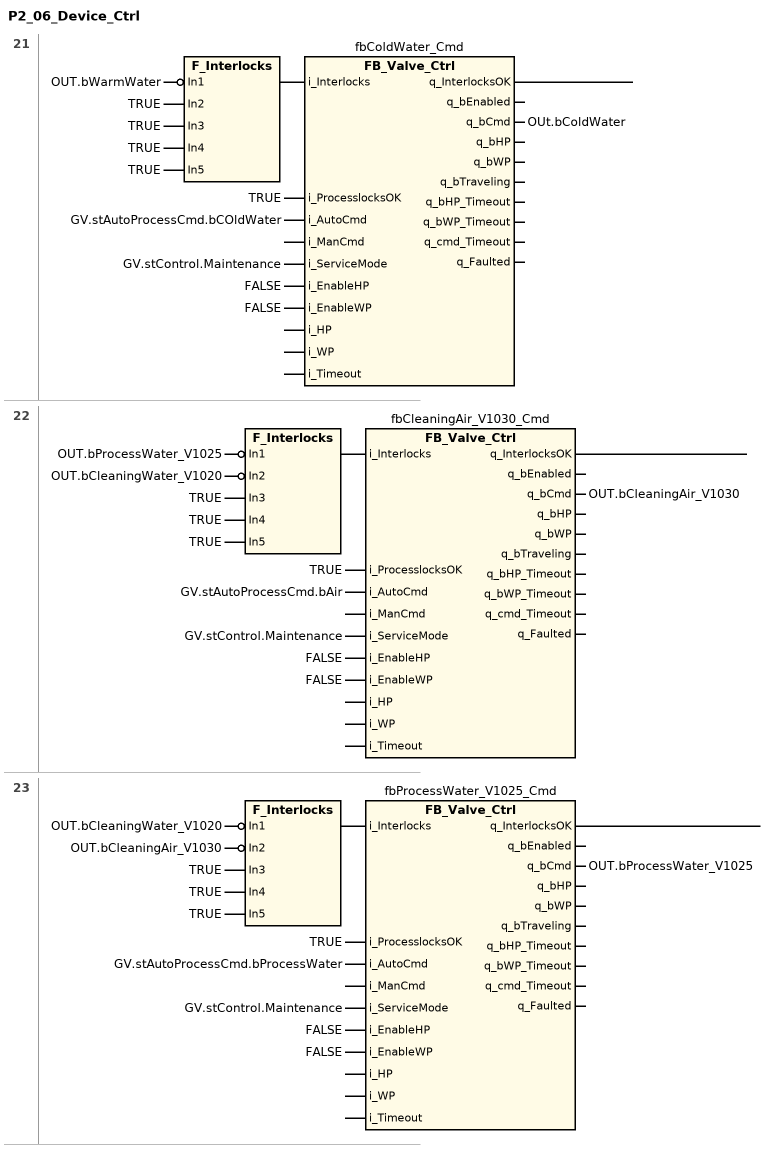
// NETWORK 21
fbColdWater_Cmd(
    i_Interlocks := F_Interlocks(In1 := NOT OUT.bWarmWater, In2 := TRUE, In3 := TRUE, In4 := TRUE, In5 := TRUE),
    i_ProcesslocksOK := TRUE,
    i_AutoCmd := GV.stAutoProcessCmd.bCOldWater,
    i_ServiceMode := GV.stControl.Maintenance,
    i_EnableHP := FALSE,
    i_EnableWP := FALSE,
    q_bCmd => OUt.bColdWater); // FB_Valve_Ctrl

// NETWORK 22
fbCleaningAir_V1030_Cmd(
    i_Interlocks := F_Interlocks(In1 := NOT OUT.bProcessWater_V1025, In2 := NOT OUT.bCleaningWater_V1020, In3 := TRUE, In4 := TRUE, In5 := TRUE),
    i_ProcesslocksOK := TRUE,
    i_AutoCmd := GV.stAutoProcessCmd.bAir,
    i_ServiceMode := GV.stControl.Maintenance,
    i_EnableHP := FALSE,
    i_EnableWP := FALSE,
    q_bCmd => OUT.bCleaningAir_V1030); // FB_Valve_Ctrl

// NETWORK 23
fbProcessWater_V1025_Cmd(
    i_Interlocks := F_Interlocks(In1 := NOT OUT.bCleaningWater_V1020, In2 := NOT OUT.bCleaningAir_V1030, In3 := TRUE, In4 := TRUE, In5 := TRUE),
    i_ProcesslocksOK := TRUE,
    i_AutoCmd := GV.stAutoProcessCmd.bProcessWater,
    i_ServiceMode := GV.stControl.Maintenance,
    i_EnableHP := FALSE,
    i_EnableWP := FALSE,
    q_bCmd => OUT.bProcessWater_V1025); // FB_Valve_Ctrl

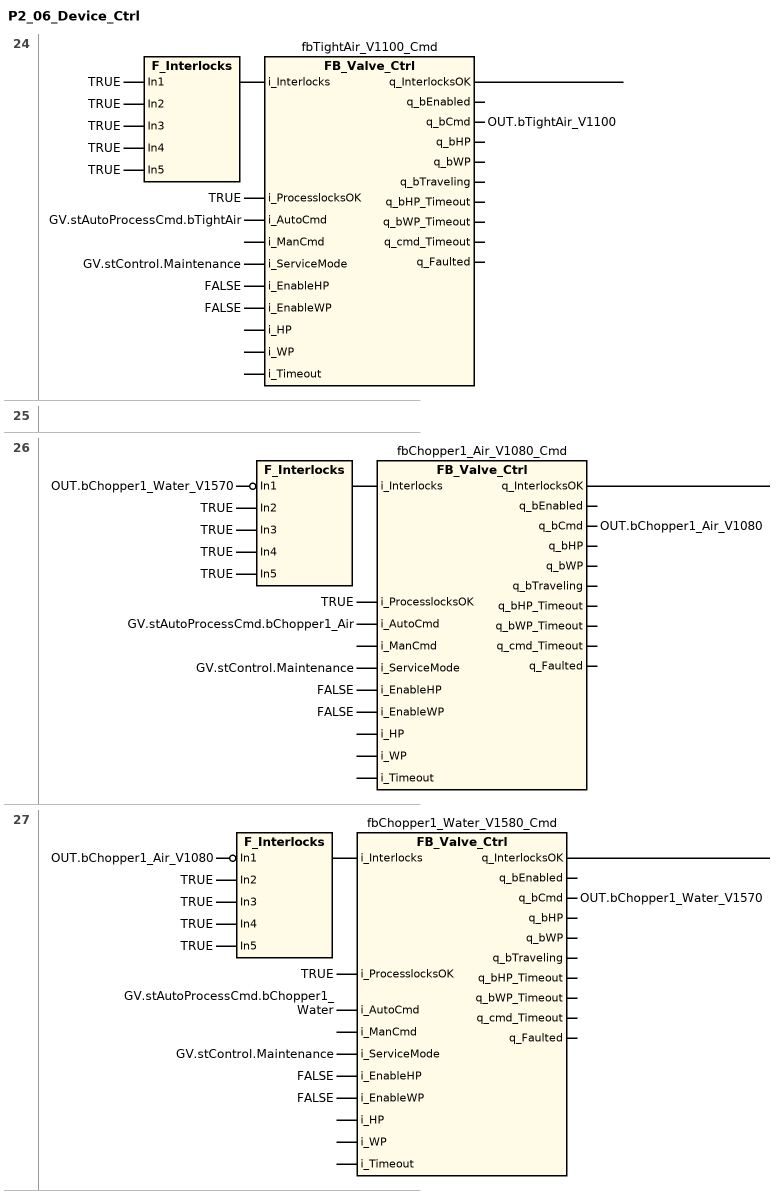
// NETWORK 24
fbTightAir_V1100_Cmd(
    i_Interlocks := F_Interlocks(In1 := TRUE, In2 := TRUE, In3 := TRUE, In4 := TRUE, In5 := TRUE),
    i_ProcesslocksOK := TRUE,
    i_AutoCmd := GV.stAutoProcessCmd.bTightAir,
    i_ServiceMode := GV.stControl.Maintenance,
    i_EnableHP := FALSE,
    i_EnableWP := FALSE,
    q_bCmd => OUT.bTightAir_V1100); // FB_Valve_Ctrl

// NETWORK 25

// NETWORK 26
fbChopper1_Air_V1080_Cmd(
    i_Interlocks := F_Interlocks(In1 := NOT OUT.bChopper1_Water_V1570, In2 := TRUE, In3 := TRUE, In4 := TRUE, In5 := TRUE),
    i_ProcesslocksOK := TRUE,
    i_AutoCmd := GV.stAutoProcessCmd.bChopper1_Air,
    i_ServiceMode := GV.stControl.Maintenance,
    i_EnableHP := FALSE,
    i_EnableWP := FALSE,
    q_bCmd => OUT.bChopper1_Air_V1080); // FB_Valve_Ctrl

// NETWORK 27
fbChopper1_Water_V1580_Cmd(
    i_Interlocks := F_Interlocks(In1 := NOT OUT.bChopper1_Air_V1080, In2 := TRUE, In3 := TRUE, In4 := TRUE, In5 := TRUE),
    i_ProcesslocksOK := TRUE,
    i_AutoCmd := GV.stAutoProcessCmd.bChopper1_Water,
    i_ServiceMode := GV.stControl.Maintenance,
    i_EnableHP := FALSE,
    i_EnableWP := FALSE,
    q_bCmd => OUT.bChopper1_Water_V1570); // FB_Valve_Ctrl

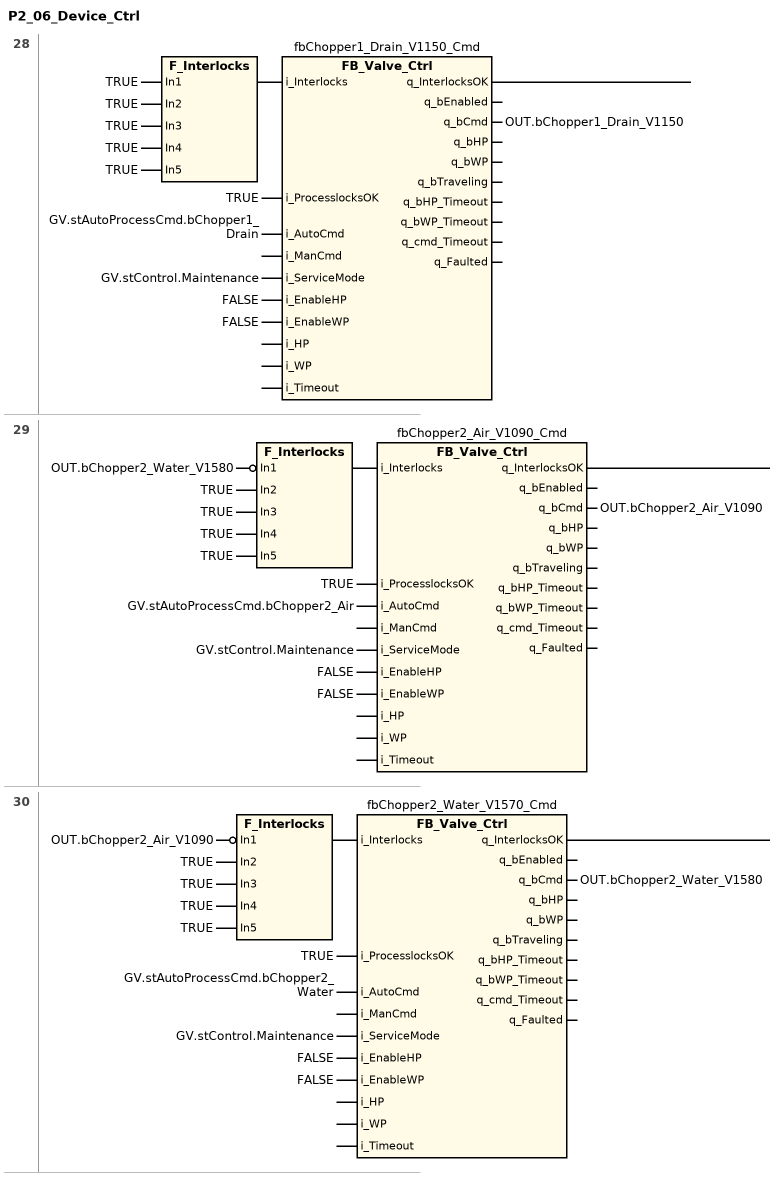
// NETWORK 28
fbChopper1_Drain_V1150_Cmd(
    i_Interlocks := F_Interlocks(In1 := TRUE, In2 := TRUE, In3 := TRUE, In4 := TRUE, In5 := TRUE),
    i_ProcesslocksOK := TRUE,
    i_AutoCmd := GV.stAutoProcessCmd.bChopper1_Drain,
    i_ServiceMode := GV.stControl.Maintenance,
    i_EnableHP := FALSE,
    i_EnableWP := FALSE,
    q_bCmd => OUT.bChopper1_Drain_V1150); // FB_Valve_Ctrl

// NETWORK 29
fbChopper2_Air_V1090_Cmd(
    i_Interlocks := F_Interlocks(In1 := NOT OUT.bChopper2_Water_V1580, In2 := TRUE, In3 := TRUE, In4 := TRUE, In5 := TRUE),
    i_ProcesslocksOK := TRUE,
    i_AutoCmd := GV.stAutoProcessCmd.bChopper2_Air,
    i_ServiceMode := GV.stControl.Maintenance,
    i_EnableHP := FALSE,
    i_EnableWP := FALSE,
    q_bCmd => OUT.bChopper2_Air_V1090); // FB_Valve_Ctrl

// NETWORK 30
fbChopper2_Water_V1570_Cmd(
    i_Interlocks := F_Interlocks(In1 := NOT OUT.bChopper2_Air_V1090, In2 := TRUE, In3 := TRUE, In4 := TRUE, In5 := TRUE),
    i_ProcesslocksOK := TRUE,
    i_AutoCmd := GV.stAutoProcessCmd.bChopper2_Water,
    i_ServiceMode := GV.stControl.Maintenance,
    i_EnableHP := FALSE,
    i_EnableWP := FALSE,
    q_bCmd => OUT.bChopper2_Water_V1580); // FB_Valve_Ctrl

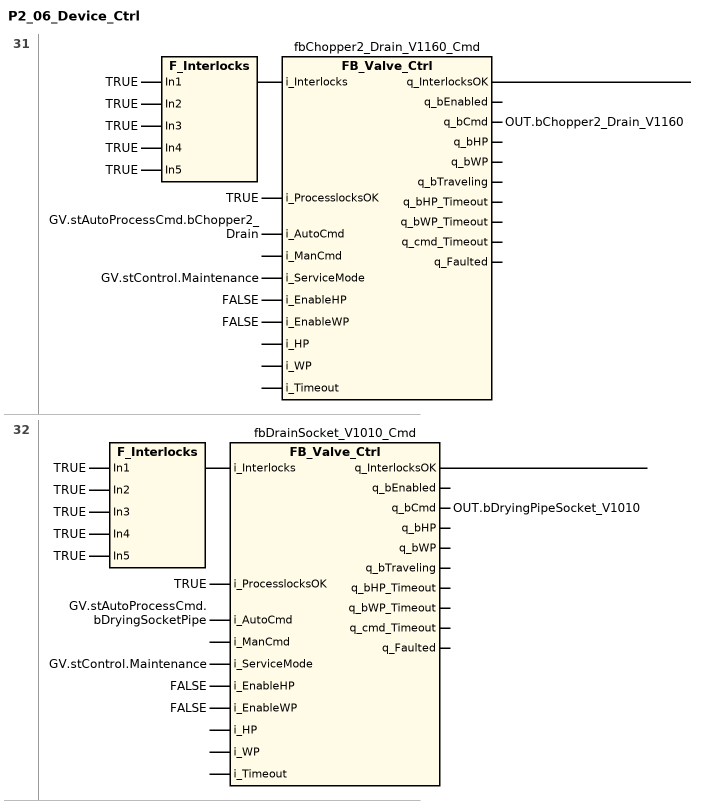
// NETWORK 31
fbChopper2_Drain_V1160_Cmd(
    i_Interlocks := F_Interlocks(In1 := TRUE, In2 := TRUE, In3 := TRUE, In4 := TRUE, In5 := TRUE),
    i_ProcesslocksOK := TRUE,
    i_AutoCmd := GV.stAutoProcessCmd.bChopper2_Drain,
    i_ServiceMode := GV.stControl.Maintenance,
    i_EnableHP := FALSE,
    i_EnableWP := FALSE,
    q_bCmd => OUT.bChopper2_Drain_V1160); // FB_Valve_Ctrl

// NETWORK 32
fbDrainSocket_V1010_Cmd(
    i_Interlocks := F_Interlocks(In1 := TRUE, In2 := TRUE, In3 := TRUE, In4 := TRUE, In5 := TRUE),
    i_ProcesslocksOK := TRUE,
    i_AutoCmd := GV.stAutoProcessCmd.bDryingSocketPipe,
    i_ServiceMode := GV.stControl.Maintenance,
    i_EnableHP := FALSE,
    i_EnableWP := FALSE,
    q_bCmd => OUT.bDryingPipeSocket_V1010); // FB_Valve_Ctrl

END_PROGRAM

// ---- FB/FB_Valve53_Ctrl.TcPOU
FUNCTION_BLOCK FB_Valve53_Ctrl
VAR_INPUT
	i_bInterlock		:BOOL;
	i_bProcesslock		:BOOL;
	i_bCmd_Disable		:BOOL;
	i_bCmd_Close		:BOOL;
	i_bCmd_HalfOpen		:BOOL;
	i_bCmd_Open			:BOOL;
	i_bSensorClosed		:BOOL;
	i_bSensorHalfOpen	:BOOL;
	i_bSensorOpen		:BOOL;
	i_tTimeout			:TIME;
	i_tTimeOutHalf		:TIME;
END_VAR
VAR_OUTPUT
	q_bCmd_Release		:BOOL;
	q_bCmd_Close		:BOOL;
	q_bCmd_Open			:BOOL;
	q_bEnabled			:BOOL;
	q_bClosed			:BOOL;
	q_bHalfOpened		:BOOL;
	q_bOpened			:BOOL;
	q_bTraveling		:BOOL;
	q_bClose_Timeout	:BOOL;
	q_bOpen_Timeout		:BOOL;
	q_bHOpen_Timeout	:BOOL;
END_VAR
VAR
	tonTimeoutClose		:TON;
	tonTimeOutHOpen		:TON;
	tonTimeoutOpen		:TON;
	bMidPosReq			:BOOL;
END_VAR
VAR // added by the converter: edge detectors and wires of the graphical bodies
    _rt1, _rt2, _rt3 : R_TRIG;
    _w1, _w2, _w3, _w4, _w5 : BOOL;
END_VAR

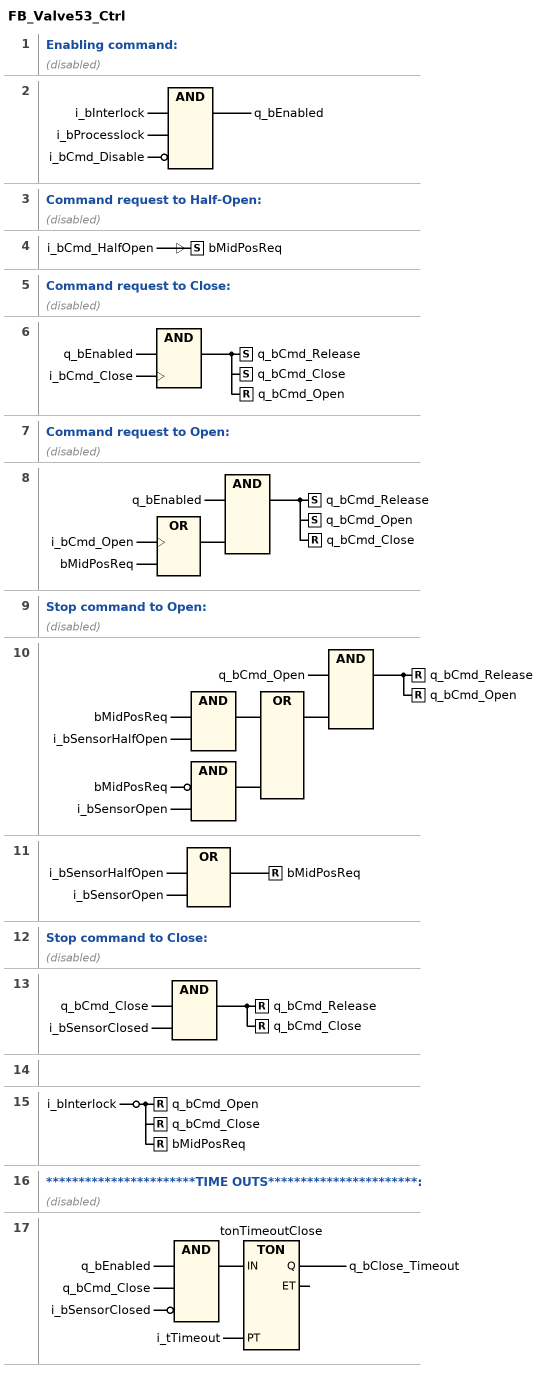
// NETWORK 1 (disabled)
// label: Enabling command

// NETWORK 2
q_bEnabled := i_bInterlock AND i_bProcesslock AND NOT i_bCmd_Disable;

// NETWORK 3 (disabled)
// label: Command request to Half-Open

// NETWORK 4
_rt1(CLK := i_bCmd_HalfOpen);
bMidPosReq S= _rt1.Q;

// NETWORK 5 (disabled)
// label: Command request to Close

// NETWORK 6
_rt2(CLK := i_bCmd_Close);
_w1 := q_bEnabled AND _rt2.Q;
q_bCmd_Release S= _w1;
q_bCmd_Close S= _w1;
q_bCmd_Open R= _w1;

// NETWORK 7 (disabled)
// label: Command request to Open

// NETWORK 8
_rt3(CLK := i_bCmd_Open);
_w2 := q_bEnabled AND (_rt3.Q OR bMidPosReq);
q_bCmd_Release S= _w2;
q_bCmd_Open S= _w2;
q_bCmd_Close R= _w2;

// NETWORK 9 (disabled)
// label: Stop command to Open

// NETWORK 10
_w3 := q_bCmd_Open AND (bMidPosReq AND i_bSensorHalfOpen OR NOT bMidPosReq AND i_bSensorOpen);
q_bCmd_Release R= _w3;
q_bCmd_Open R= _w3;

// NETWORK 11
bMidPosReq R= i_bSensorHalfOpen OR i_bSensorOpen;

// NETWORK 12 (disabled)
// label: Stop command to Close

// NETWORK 13
_w4 := q_bCmd_Close AND i_bSensorClosed;
q_bCmd_Release R= _w4;
q_bCmd_Close R= _w4;

// NETWORK 14

// NETWORK 15
_w5 := NOT i_bInterlock;
q_bCmd_Open R= _w5;
q_bCmd_Close R= _w5;
bMidPosReq R= _w5;

// NETWORK 16 (disabled)
// label: ***********************TIME OUTS***********************

// NETWORK 17
tonTimeoutClose(IN := q_bEnabled AND q_bCmd_Close AND NOT i_bSensorClosed, PT := i_tTimeout); // TON
q_bClose_Timeout := tonTimeoutClose.Q;

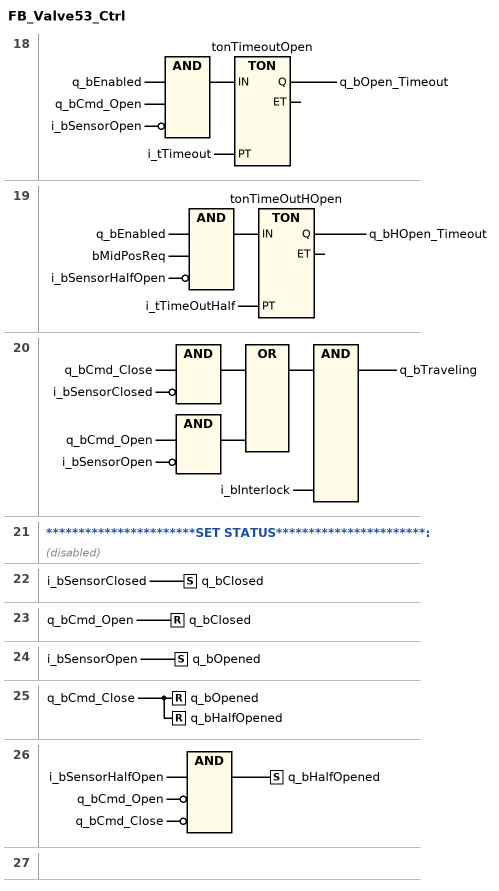
// NETWORK 18
tonTimeoutOpen(IN := q_bEnabled AND q_bCmd_Open AND NOT i_bSensorOpen, PT := i_tTimeout); // TON
q_bOpen_Timeout := tonTimeoutOpen.Q;

// NETWORK 19
tonTimeOutHOpen(IN := q_bEnabled AND bMidPosReq AND NOT i_bSensorHalfOpen, PT := i_tTimeOutHalf); // TON
q_bHOpen_Timeout := tonTimeOutHOpen.Q;

// NETWORK 20
q_bTraveling := (q_bCmd_Close AND NOT i_bSensorClosed OR q_bCmd_Open AND NOT i_bSensorOpen) AND i_bInterlock;

// NETWORK 21 (disabled)
// label: ***********************SET STATUS***********************

// NETWORK 22
q_bClosed S= i_bSensorClosed;

// NETWORK 23
q_bClosed R= q_bCmd_Open;

// NETWORK 24
q_bOpened S= i_bSensorOpen;

// NETWORK 25
q_bOpened R= q_bCmd_Close;
q_bHalfOpened R= q_bCmd_Close;

// NETWORK 26
q_bHalfOpened S= i_bSensorHalfOpen AND NOT q_bCmd_Open AND NOT q_bCmd_Close;

// NETWORK 27

END_FUNCTION_BLOCK

// ---- FB/FB_Mixer_Ctrl.TcPOU
FUNCTION_BLOCK FB_Mixer_Ctrl
VAR_INPUT
	i_Interlocks		:ARRAY[1..5] OF BOOL;
	i_AutoCmdFwd		:BOOL;
	i_AutoCmdBcw		:BOOL;
	i_AutoSpeedSP		:REAL;
	i_ManCmdFwd			:BOOL;
	i_ManCmdBcw			:BOOL;
	i_ManStop			:BOOL;
	i_ManSpeedSP		:REAL;
	i_SpeedAP			:REAL;
	i_CurrentAP			:REAL;
	i_ServiceMode		:BOOL;
END_VAR
VAR_OUTPUT
	q_InterlocksOK		:BOOL;
	q_bCmdFwd			:BOOL;
	q_bCmdBcw			:BOOL;
	q_rSpeedSP			:REAL;
END_VAR
VAR
	bCmdFwd				:BOOL;
	bCmdBcw				:BOOL;
	tofCMDFwd			:TOF;
	tofCMDBcw			:TOF;
	tonFwdOff			:TON;
	tonBcwOff			:TON;
END_VAR
VAR // added by the converter: edge detectors and wires of the graphical bodies
    _w1 : BOOL;
END_VAR

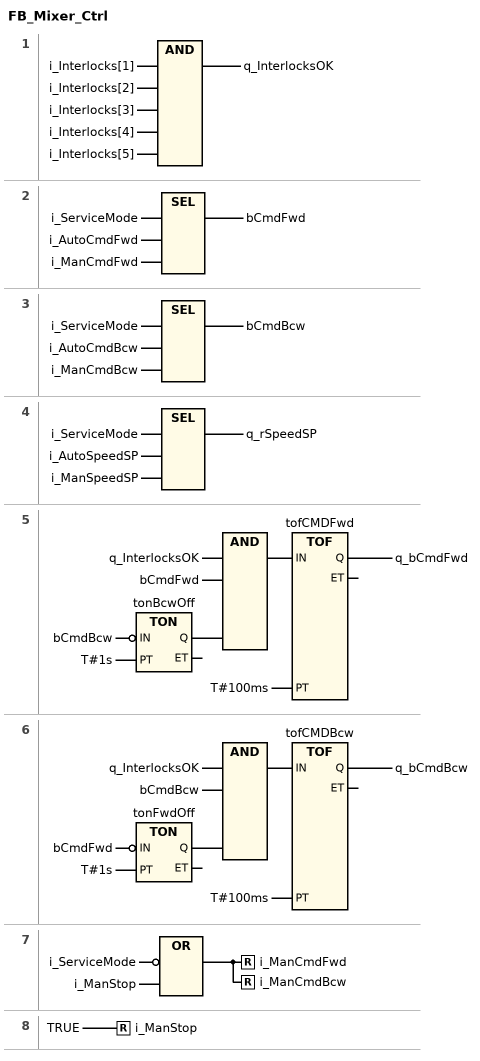
// NETWORK 1
q_InterlocksOK := i_Interlocks[1] AND i_Interlocks[2] AND i_Interlocks[3] AND i_Interlocks[4] AND i_Interlocks[5];

// NETWORK 2
bCmdFwd := SEL(i_ServiceMode, i_AutoCmdFwd, i_ManCmdFwd);

// NETWORK 3
bCmdBcw := SEL(i_ServiceMode, i_AutoCmdBcw, i_ManCmdBcw);

// NETWORK 4
q_rSpeedSP := SEL(i_ServiceMode, i_AutoSpeedSP, i_ManSpeedSP);

// NETWORK 5
tonBcwOff(IN := NOT bCmdBcw, PT := T#1s); // TON
tofCMDFwd(IN := q_InterlocksOK AND bCmdFwd AND tonBcwOff.Q, PT := T#100ms); // TOF
q_bCmdFwd := tofCMDFwd.Q;

// NETWORK 6
tonFwdOff(IN := NOT bCmdFwd, PT := T#1s); // TON
tofCMDBcw(IN := q_InterlocksOK AND bCmdBcw AND tonFwdOff.Q, PT := T#100ms); // TOF
q_bCmdBcw := tofCMDBcw.Q;

// NETWORK 7
_w1 := NOT i_ServiceMode OR i_ManStop;
i_ManCmdFwd R= _w1;
i_ManCmdBcw R= _w1;

// NETWORK 8
i_ManStop R= TRUE;

END_FUNCTION_BLOCK

// ---- FB/FB_AnalogOutput.TcPOU
// Created by Dimitar Stojanov 06.2023 

//Functionality: Use this block to scale Analog Outputs

FUNCTION_BLOCK FB_AnalogOutput
VAR_INPUT
	i_rValue 							:REAL;
	i_rData_Low 						:REAL;
	i_rData_High 						:REAL;
	i_rScaled_Low						:INT	:=0;
	i_rScaled_High						:INT	:=32676;
	i_iOffset 							:INT;
	
END_VAR
VAR_OUTPUT
	q_iScaled							:INT;
END_VAR
VAR
	K								    :REAL;
END_VAR

K := ((i_rScaled_High - i_rScaled_Low) / (i_rData_High - i_rData_Low));
q_iScaled:=REAL_TO_INT((K * i_rValue) + i_iOffset);

END_FUNCTION_BLOCK

// ---- FB/FB_Chopper_Ctrl.TcPOU
FUNCTION_BLOCK FB_Chopper_Ctrl
VAR_INPUT
	i_Interlocks		:ARRAY[1..5] OF BOOL;
	i_AutoSlowCmd		:BOOL;
	i_AutoFastCmd		:BOOL;
	i_ManSlowCmd		:BOOL;
	i_ManFastCmd		:BOOL;
	I_ManStop			:BOOL;
	i_rSpeed			:REAL;
	i_ServiceMode		:BOOL;
END_VAR
VAR_OUTPUT
	q_InterlocksOK		:BOOL;
	q_bCmdFast			:BOOL;
	q_bCmdSlow			:BOOL;
	q_rSpeed			:REAL;
END_VAR
VAR
	bCmdSlow			:BOOL;
	bCmdFast			:BOOL;
	tofSlowCMD			:TOF;
	tofFastCMD			:TOF;
	tonSlowOff			:TON;
	tonFastOff			:TON;
END_VAR
VAR // added by the converter: edge detectors and wires of the graphical bodies
    _w1 : BOOL;
END_VAR

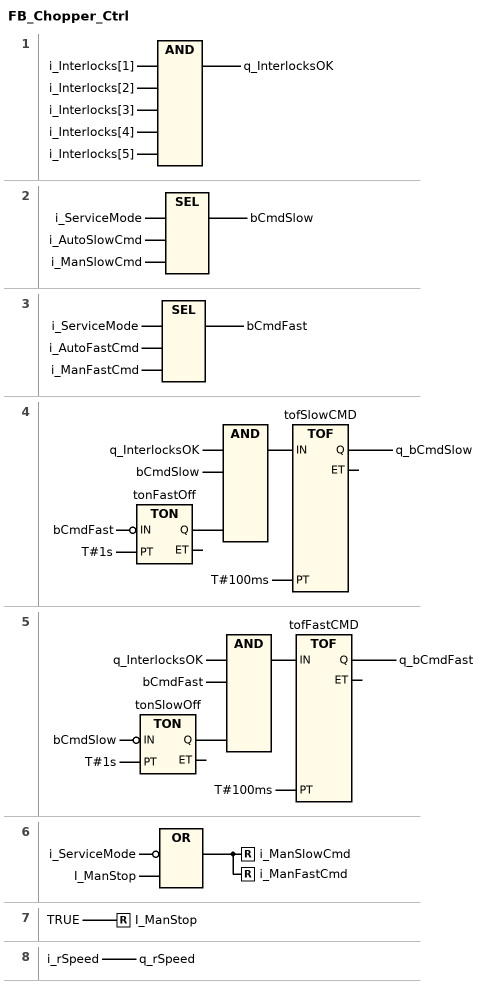
// NETWORK 1
q_InterlocksOK := i_Interlocks[1] AND i_Interlocks[2] AND i_Interlocks[3] AND i_Interlocks[4] AND i_Interlocks[5];

// NETWORK 2
bCmdSlow := SEL(i_ServiceMode, i_AutoSlowCmd, i_ManSlowCmd);

// NETWORK 3
bCmdFast := SEL(i_ServiceMode, i_AutoFastCmd, i_ManFastCmd);

// NETWORK 4
tonFastOff(IN := NOT bCmdFast, PT := T#1s); // TON
tofSlowCMD(IN := q_InterlocksOK AND bCmdSlow AND tonFastOff.Q, PT := T#100ms); // TOF
q_bCmdSlow := tofSlowCMD.Q;

// NETWORK 5
tonSlowOff(IN := NOT bCmdSlow, PT := T#1s); // TON
tofFastCMD(IN := q_InterlocksOK AND bCmdFast AND tonSlowOff.Q, PT := T#100ms); // TOF
q_bCmdFast := tofFastCMD.Q;

// NETWORK 6
_w1 := NOT i_ServiceMode OR I_ManStop;
i_ManSlowCmd R= _w1;
i_ManFastCmd R= _w1;

// NETWORK 7
I_ManStop R= TRUE;

// NETWORK 8
q_rSpeed := i_rSpeed;

END_FUNCTION_BLOCK

// ---- FB/FB_Valve_Ctrl.TcPOU
FUNCTION_BLOCK FB_Valve_Ctrl
VAR_INPUT
	i_Interlocks		:ARRAY[1..5] OF BOOL;
	i_ProcesslocksOK	:BOOL;
	i_AutoCmd			:BOOL;
	i_ManCmd			:BOOL;
	i_ServiceMode		:BOOL;
	i_EnableHP			:BOOL;
	i_EnableWP			:BOOL;
	i_HP				:BOOL;
	i_WP				:BOOL;
	i_Timeout			:TIME;
END_VAR
VAR_OUTPUT
	q_InterlocksOK		:BOOL;
	q_bEnabled			:BOOL;
	q_bCmd				:BOOL;
	q_bHP				:BOOL;
	q_bWP				:BOOL;
	q_bTraveling		:BOOL;
	q_bHP_Timeout		:BOOL;
	q_bWP_Timeout		:BOOL;
	q_cmd_Timeout		:BOOL;
	q_Faulted			:BOOL;
END_VAR
VAR
	tonTimeoutHP		:TON;
	tonTimeoutWP		:TON;
	tonTimeoutCmd		:TON;
	tofDelayOut			:TOF;
	bCmd				:BOOL;
END_VAR

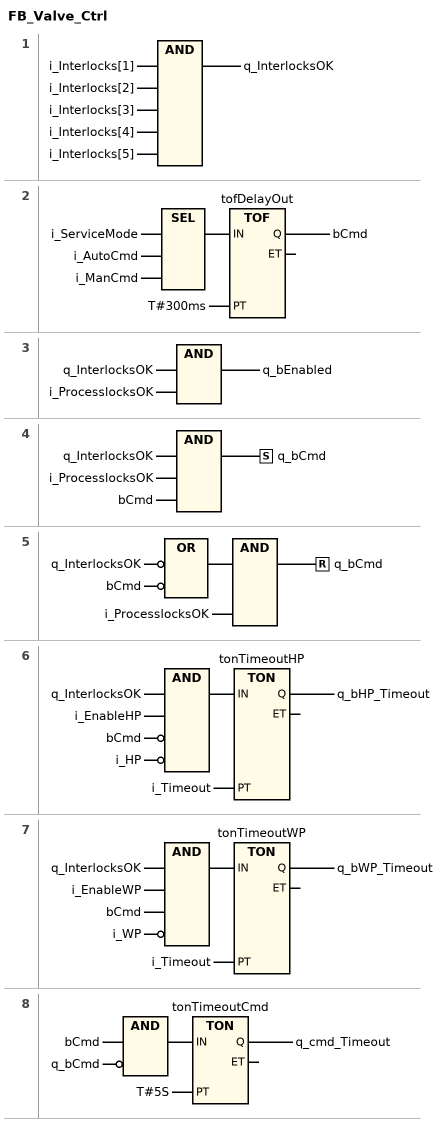
// NETWORK 1
q_InterlocksOK := i_Interlocks[1] AND i_Interlocks[2] AND i_Interlocks[3] AND i_Interlocks[4] AND i_Interlocks[5];

// NETWORK 2
tofDelayOut(IN := SEL(i_ServiceMode, i_AutoCmd, i_ManCmd), PT := T#300ms); // TOF
bCmd := tofDelayOut.Q;

// NETWORK 3
q_bEnabled := q_InterlocksOK AND i_ProcesslocksOK;

// NETWORK 4
q_bCmd S= q_InterlocksOK AND i_ProcesslocksOK AND bCmd;

// NETWORK 5
q_bCmd R= (NOT q_InterlocksOK OR NOT bCmd) AND i_ProcesslocksOK;

// NETWORK 6
tonTimeoutHP(IN := q_InterlocksOK AND i_EnableHP AND NOT bCmd AND NOT i_HP, PT := i_Timeout); // TON
q_bHP_Timeout := tonTimeoutHP.Q;

// NETWORK 7
tonTimeoutWP(IN := q_InterlocksOK AND i_EnableWP AND bCmd AND NOT i_WP, PT := i_Timeout); // TON
q_bWP_Timeout := tonTimeoutWP.Q;

// NETWORK 8
tonTimeoutCmd(IN := bCmd AND NOT q_bCmd, PT := T#5S); // TON
q_cmd_Timeout := tonTimeoutCmd.Q;

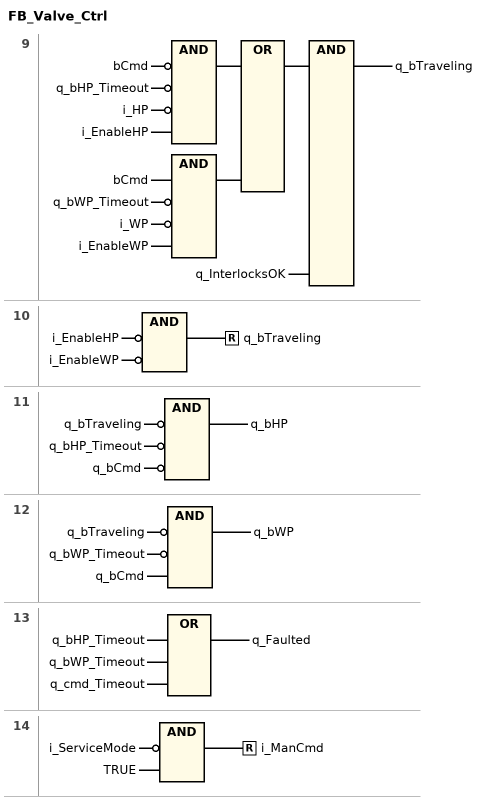
// NETWORK 9
q_bTraveling := (NOT bCmd AND NOT q_bHP_Timeout AND NOT i_HP AND i_EnableHP OR bCmd AND NOT q_bWP_Timeout AND NOT i_WP AND i_EnableWP) AND q_InterlocksOK;

// NETWORK 10
q_bTraveling R= NOT i_EnableHP AND NOT i_EnableWP;

// NETWORK 11
q_bHP := NOT q_bTraveling AND NOT q_bHP_Timeout AND NOT q_bCmd;

// NETWORK 12
q_bWP := NOT q_bTraveling AND NOT q_bWP_Timeout AND q_bCmd;

// NETWORK 13
q_Faulted := q_bHP_Timeout OR q_bWP_Timeout OR q_cmd_Timeout;

// NETWORK 14
i_ManCmd R= NOT i_ServiceMode AND TRUE;

END_FUNCTION_BLOCK

// ---- POUs/2. Process/Production/_Discharging.TcPOU
PROGRAM _Discharging
VAR_INPUT
	i_bStart							:BOOL;
	i_bProcessFinished					:BOOL;
	i_bStepFinished						:BOOL;
	i_bSkipStep							:BOOL;
	i_bBarrelInPos						:BOOL;
	i_bManualFlapOpen					:BOOL;
	i_bManualFlapClose					:BOOL;
	i_iMixer							:INT;
	i_rMixerSpeed						:REAL;
	i_bMixerStart						:BOOL; 	
	i_iChopper							:INT;	
END_VAR
VAR
	iStep						:INT;
	iPrevStep					:INT;
	Seq_TON						:ARRAY[0..9] OF TON;
	Seq_Time					:ARRAY[0..9] OF TIME;
	trigMixer					:R_TRIG;
	bStartMixer					:BOOL;
	tonStepTime					:TON;
END_VAR
VAR_OUTPUT
	q_bRunning						:BOOL;
	q_bFinished						:BOOL;
	q_stCmd							:ST_ProcessCmd;
	q_bDisOpenReq					:BOOL;
	q_bDischargeCmdEnable			:BOOL;
	q_bBarrelInPosReq				:BOOL;
	q_tStepTime						:TIME;
END_VAR

trigMixer(CLK:=i_bMixerStart);


q_bRunning:=iStep<>0;

IF i_bSkipStep THEN
	iStep:=1000;
END_IF

IF NOT i_bStart THEN
	iStep:=0;
END_IF

CASE iStep OF
	0:
		IF i_bStart THEN
			q_bFinished:=FALSE;
			iStep:=40;
		END_IF
		
		IF iStep <> 0 THEN
			iPrevStep:=0;
		END_IF
		
	40:
		IF i_bBarrelInPos THEN
			iStep:=50;
		END_IF
		
	50:
		IF i_bManualFlapOpen THEN
			iStep:=100;
		END_IF
		
		IF iStep <> 50 THEN
			iPrevStep:=50;
		END_IF
	
	100:
		
		IF i_bProcessFinished THEN
			iStep:=1000;
		END_IF
		IF iStep <> 100 THEN
			iPrevStep:=100;
		END_IF

		
	1000:
		q_bFinished:=TRUE;
		IF i_bStepFinished THEN
			iStep:=0;
		END_IF
END_CASE

IF trigMixer.Q THEN
	bStartMixer:= NOT bStartMixer;
END_IF

q_bBarrelInPosReq:=F_StepCMP(iStep,40,0,0,0,0,0,0,0,0,0);

q_bDisOpenReq:=F_StepCMP(iStep,50,0,0,0,0,0,0,0,0,0);
IF F_StepCMP(iStep,50,0,0,0,0,0,0,0,0,0) THEN
	q_stCmd.bDischargeClose:=FALSE;
	q_stCmd.bDischargeOpen:=TRUE;
ELSE
	q_stCmd.bDischargeClose:=FALSE;
	q_stCmd.bDischargeOpen:=FALSE;
END_IF

q_bDischargeCmdEnable:=F_StepCMP(iStep,100,0,0,0,0,0,0,0,0,0);

IF F_StepCMP(iStep,100,0,0,0,0,0,0,0,0,0) AND bStartMixer THEN
	q_stCmd.iMixer:=i_iMixer;
	q_stCmd.rMixerSpeed:=i_rMixerSpeed;
ELSE
	q_stCmd.iMixer:=0;
	q_stCmd.rMixerSpeed:=0;
	bStartMixer:=FALSE;
END_IF

IF F_StepCMP(iStep,100,0,0,0,0,0,0,0,0,0) AND bStartMixer THEN
	q_stCmd.iChopper:=i_iChopper;
ELSE
	q_stCmd.iChopper:=0;
END_IF

q_stCmd.bTightAir:=F_StepCMP(iStep,50,100,0,0,0,0,0,0,0,0);
q_stCmd.bChopper1_Air:=F_StepCMP(iStep,50,100,0,0,0,0,0,0,0,0);
q_stCmd.bChopper2_Air:=F_StepCMP(iStep,50,100,0,0,0,0,0,0,0,0);

//Statistic and Status
tonStepTime(IN:=q_bRunning,PT:=T#5H);
q_tStepTime:=tonStepTime.ET;

END_PROGRAM

// ---- FB/F_StepCMP.TcPOU
FUNCTION F_StepCMP : BOOL
VAR_INPUT
	iStep			:INT:=0;
	i1				:INT:=0;
	i2				:INT:=0;
	i3				:INT:=0;
	i4				:INT:=0;
	i5				:INT:=0;
	i6				:INT:=0;
	i7				:INT:=0;
	i8				:INT:=0;
	i9				:INT:=0;
	i10				:INT:=0;
END_VAR

F_StepCMP:=((iStep=i1) OR 
			(iStep=i2) OR 
			(iStep=i3) OR 
			(iStep=i4) OR 
			(iStep=i5) OR 
			(iStep=i6) OR 
			(iStep=i7) OR 
			(iStep=i8) OR 
			(iStep=i9) OR 
			(iStep=i10)) AND
			(iStep<>0);

END_FUNCTION

// ---- FB/F_Interlocks.TcPOU
FUNCTION F_Interlocks : ARRAY[1..5] OF BOOL
VAR_INPUT
	In1		:BOOL;
	In2		:BOOL;
	In3		:BOOL;
	In4		:BOOL;
	In5		:BOOL;
END_VAR
VAR
END_VAR

F_Interlocks[1] := In1;
F_Interlocks[2] := In2;
F_Interlocks[3] := In3;
F_Interlocks[4] := In4;
F_Interlocks[5] := In5;

END_FUNCTION

// ---- POUs/3. Report/P3_06_CreateReport.TcPOU
PROGRAM P3_06_CreateReport
VAR
	iStep					:INT;
	iError					:INT;
	tonResetError			:TON;
	trigStart				:R_TRIG;
	tonDelayStart			:TON;
	
	
	
	fbReport				:FB_PythonScript;
	fbSettingDelete			:FB_FileDelete;
	fbRecipeDelete			:FB_FileDelete;
	fbDeleteOldestBatch		:FB_DeleteOldestFile;
	fbSaveAsAlarm			:FB_FileSaveAs;
END_VAR


VAR PERSISTENT
	iReportsCreated			:INT;
END_VAR

ACT_CMDs();
tonResetError(IN:=(iError<>0),PT:=T#3S);
IF tonResetError.Q THEN
	iError:=0;
END_IF

trigStart(CLK:=GV.bBatchClose);

tonDelayStart(IN:=(iStep=10),PT:=T#1S);
CASE iStep OF
	
	0:
		IF trigStart.Q THEN
			iError:=0;
			iStep:=10;
		END_IF
		
	10:
		IF tonDelayStart.Q THEN
			iStep:=20;
		END_IF
		
	20:
		GV.stReport.bExport_Alarms:=TRUE;
		iStep:=25;
	25:
		IF NOT GV.stReport.bExport_Alarms THEN
			iStep:=30;
		END_IF
	26:
		GV.stReport.bSaveAs_Alarms:=TRUE;
		iStep:=27;
	27:
		IF NOT fbSaveAsAlarm.q_bBusy THEN
			iStep:=30;
		END_IF
		
	30:
		GV.stReport.bCreate_Report:=TRUE;
		IF fbReport.q_bBusy THEN
			iStep:=35;
		END_IF
	35:
		IF NOT fbReport.q_bBusy AND fbReport.q_bDone THEN
			iStep:=40;
		ELSIF fbReport.q_bError THEN
			iError:=iStep;
			iStep:=999;
		END_IF
	40:
		GV.stReport.bDelete_Data:=TRUE;
		iStep:=45;
	45:
		IF NOT GV.stReport.bDelete_Data THEN
			iStep:=50;
		END_IF
		
	50:
		GV.stReport.bDelete_OldestReport:=TRUE;
		IF fbDeleteOldestBatch.q_bBusy THEN
			iStep:=55;
		END_IF
	55:
		IF NOT fbDeleteOldestBatch.q_bBusy AND fbDeleteOldestBatch.q_bDone THEN
			iStep:=900;
		ELSIF fbDeleteOldestBatch.q_bError THEN
			iStep:=900;
			iError:=iStep;
		END_IF
		
	900:
		iReportsCreated:=iReportsCreated+1;
		GV.stReport.bStartSend_Sequence:=TRUE;
		iStep:=0;
	999:
		iStep:=0;
END_CASE

ACTION ACT_CMDs:
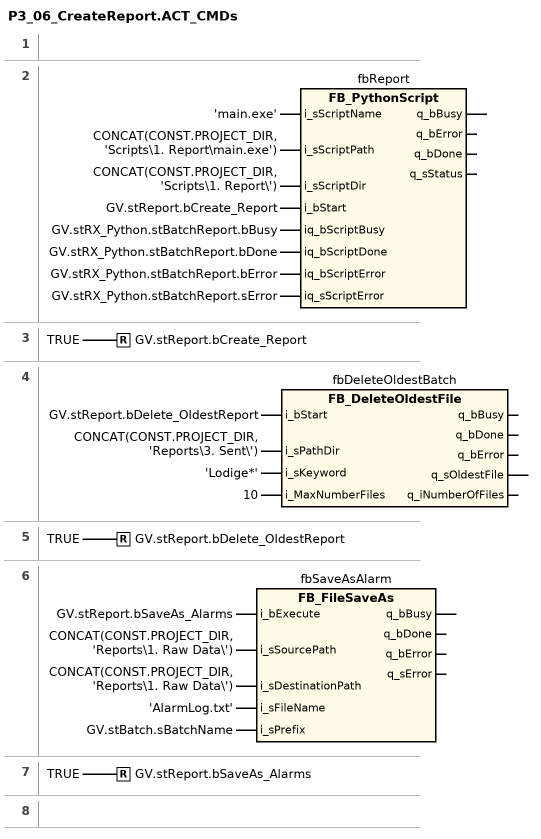
// NETWORK 1

// NETWORK 2
fbReport(
    i_sScriptName := 'main.exe',
    i_sScriptPath := CONCAT(CONST.PROJECT_DIR,'Scripts\1. Report\main.exe'),
    i_sScriptDir := CONCAT(CONST.PROJECT_DIR,'Scripts\1. Report\'),
    i_bStart := GV.stReport.bCreate_Report,
    iq_bScriptBusy := GV.stRX_Python.stBatchReport.bBusy,
    iq_bScriptDone := GV.stRX_Python.stBatchReport.bDone,
    iq_bScriptError := GV.stRX_Python.stBatchReport.bError,
    iq_sScriptError := GV.stRX_Python.stBatchReport.sError); // FB_PythonScript

// NETWORK 3
GV.stReport.bCreate_Report R= TRUE;

// NETWORK 4
fbDeleteOldestBatch(
    i_bStart := GV.stReport.bDelete_OldestReport,
    i_sPathDir := CONCAT(CONST.PROJECT_DIR,'Reports\3. Sent\'),
    i_sKeyword := 'Lodige*',
    i_MaxNumberFiles := 10); // FB_DeleteOldestFile

// NETWORK 5
GV.stReport.bDelete_OldestReport R= TRUE;

// NETWORK 6
fbSaveAsAlarm(
    i_bExecute := GV.stReport.bSaveAs_Alarms,
    i_sSourcePath := CONCAT(CONST.PROJECT_DIR,'Reports\1. Raw Data\'),
    i_sDestinationPath := CONCAT(CONST.PROJECT_DIR,'Reports\1. Raw Data\'),
    i_sFileName := 'AlarmLog.txt',
    i_sPrefix := GV.stBatch.sBatchName); // FB_FileSaveAs

// NETWORK 7
GV.stReport.bSaveAs_Alarms R= TRUE;

// NETWORK 8
END_ACTION

END_PROGRAM

// ---- FB/FB_PythonScript.TcPOU
FUNCTION_BLOCK FB_PythonScript
VAR_INPUT
	i_sScriptName		:STRING;
	i_sScriptPath		:STRING;
	i_sScriptDir		:STRING;
	i_bStart			:BOOL;
END_VAR
VAR_IN_OUT
	iq_bScriptBusy		:BOOL;
	iq_bScriptDone		:BOOL;
	iq_bScriptError		:BOOL;
	iq_sScriptError		:STRING;
END_VAR
VAR_OUTPUT
	q_bBusy				:BOOL;
	q_bError			:BOOL;
	q_bDone				:BOOL;
	q_sStatus			:STRING;
END_VAR
VAR
	ntProcess			:NT_StartProcess;
	bStartNT			:BOOL;

	iStep				:INT;
	tTimeOut_TON1		:TON;
	tTimeOut1			:TIME;
	tTimeOut_TON2		:TON;
	tTimeOut2			:TIME;
END_VAR

ACT_StartProcess();

tTimeOut1:=T#30S;
tTimeOut2:=T#30S;

q_sStatus:=iq_sScriptError;

CASE iStep OF
	
	0:

		q_bBusy:=FALSE;
		tTimeOut_TON1(IN:=FALSE,PT:=tTimeOut1);
		tTimeOut_TON2(IN:=FALSE,PT:=tTimeOut2);
	
		IF i_bStart THEN
			q_bError:=FALSE;
			q_bDone:=FALSE;
			q_bBusy:=TRUE;
			
			iq_bScriptBusy:=FALSE;
			iq_bScriptDone:=FALSE;
			iq_bScriptError:=FALSE;
			iq_sScriptError:='';
			
			iStep:=10;
		END_IF
	
	10:
		bStartNT:=TRUE;
		IF ntProcess.BUSY THEN
			iStep:=15;
		END_IF
	
	15:
		IF NOT ntProcess.BUSY THEN
			iStep:=20;
		ELSIF ntProcess.ERR THEN
			iStep:=999;
		END_IF
	20:
		tTimeOut_TON1(IN:=TRUE,PT:=tTimeOut1);
		IF NOT iq_bScriptDone AND NOT iq_bScriptError THEN
			iStep:=30;
		ELSIF tTimeOut_TON1.Q OR iq_bScriptError THEN
			iStep:=999;
		END_IF
	30:
		tTimeOut_TON2(IN:=TRUE,PT:=tTimeOut2);
		IF iq_bScriptDone AND NOT iq_bScriptError THEN 
			iStep:=50;	
		ELSIF tTimeOut_TON2.Q OR iq_bScriptError THEN
			iStep:=999;
		END_IF
		
	50:
		q_bDone:=TRUE;
		iStep:=0;
	999:
		
		q_bError:=TRUE;
		iStep:=0;
		
		
END_CASE

ACTION ACT_StartProcess:
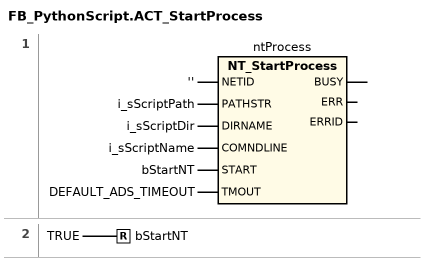
// NETWORK 1
ntProcess(
    NETID := '',
    PATHSTR := i_sScriptPath,
    DIRNAME := i_sScriptDir,
    COMNDLINE := i_sScriptName,
    START := bStartNT,
    TMOUT := DEFAULT_ADS_TIMEOUT); // NT_StartProcess

// NETWORK 2
bStartNT R= TRUE;
END_ACTION

END_FUNCTION_BLOCK

// ---- FB/FB_DeleteOldestFile.TcPOU
FUNCTION_BLOCK FB_DeleteOldestFile
VAR_INPUT
	i_bStart					:BOOL;
	i_sPathDir					:STRING[300];
	i_sKeyword					:STRING:='*';
	i_MaxNumberFiles			:UINT;
END_VAR
VAR_OUTPUT
	q_bBusy							:BOOL;
	q_bDone							:BOOL;
	q_bError						:BOOL;
	q_sOldestFile					:STRING;
	q_iNumberOfFiles				:UINT;
	
END_VAR
VAR
	fbFindFile				:FB_EnumFindFileEntry;
	eCmd					:E_EnumCmdType;
	bExecute				:BOOL;
	stFindFile				:ST_FindFileEntry;
	fbFileDelete			:FB_FileDelete;
	iStep					:INT:=0;
	sPath					:STRING[300];
	bDelete					:BOOL;
	sDeletePath				:STRING[300];
END_VAR

sPath:=CONCAT(i_sPathDir,i_sKeyword);
ACT_Files();
CASE iStep OF
	0:
		q_bBusy:=FALSE;
		IF i_bStart THEN
			q_iNumberOfFiles:=0;
			q_bDone:=FALSE;
			q_bError:=FALSE;
			q_bBusy:=TRUE;
			iStep:=10;
		END_IF
		
	10:
		eCmd := 0;
		bExecute:=TRUE;
		IF fbFindFile.bBusy THEN
			iStep:=20;
		END_IF
		
	20:
		IF NOT fbFindFile.bBusy THEN
			IF NOT fbFindFile.bError AND NOT fbFindFile.bEOE THEN
				q_sOldestFile:=stFindFile.sFileName;
				bExecute:=FALSE;
				iStep:=30;
			ELSIF NOT fbFindFile.bError AND fbFindFile.bEOE THEN
				bExecute:=FALSE;
				iStep:=100;
			ELSIF fbFindFile.bError THEN
				iStep:=999;
			END_IF
		END_IF
		
	30:
		q_iNumberOfFiles:=q_iNumberOfFiles+1;
		iStep:=40;
	
	40:
		eCmd := 1;
		bExecute:=TRUE;
		IF fbFindFile.bBusy THEN
			iStep:=50;
		END_IF
	
	50:
		IF NOT fbFindFile.bBusy THEN
			IF NOT fbFindFile.bError AND NOT fbFindFile.bEOE THEN
				bExecute:=FALSE;
				iStep:=30;
			ELSIF NOT fbFindFile.bError AND fbFindFile.bEOE THEN
				bExecute:=FALSE;
				iStep:=100;
			ELSIF fbFindFile.bError THEN
				iStep:=999;
			END_IF
		END_IF
		
	100:
		eCmd:=2;
		bExecute:=TRUE;
		IF NOT fbFindFile.bBusy THEN
			iStep:=150;
		END_IF
		
	150:
		IF q_iNumberOfFiles >= i_MaxNumberFiles THEN
			iStep:=200;
		ELSE
			iStep:=300;
		END_IF
		
	200:
		sDeletePath:=CONCAT(i_sPathDir,q_sOldestFile);
		bDelete:=TRUE;
		iStep:=210;
	
	210:
		IF NOT fbFileDelete.bBusy THEN
			iStep:=300;
		END_IF
		
	300:
		q_bDone:=TRUE;
		iStep:=0;
		
	999:
		q_bError:=TRUE;
		iStep:=0;
		
		
END_CASE

ACTION ACT_Files:
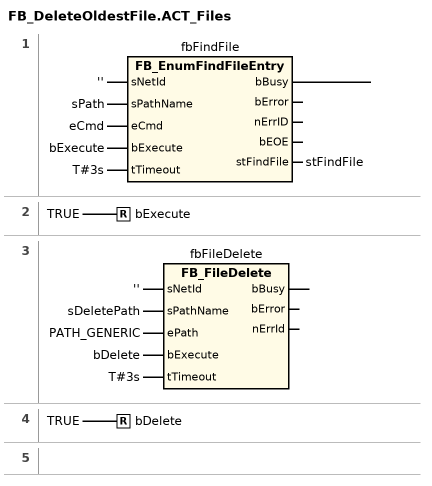
// NETWORK 1
fbFindFile(
    sNetId := '',
    sPathName := sPath,
    eCmd := eCmd,
    bExecute := bExecute,
    tTimeout := T#3s,
    stFindFile => stFindFile); // FB_EnumFindFileEntry

// NETWORK 2
bExecute R= TRUE;

// NETWORK 3
fbFileDelete(
    sNetId := '',
    sPathName := sDeletePath,
    ePath := PATH_GENERIC,
    bExecute := bDelete,
    tTimeout := T#3s); // FB_FileDelete

// NETWORK 4
bDelete R= TRUE;

// NETWORK 5
END_ACTION

END_FUNCTION_BLOCK

// ---- FB/FB_FileSaveAs.TcPOU
FUNCTION_BLOCK FB_FileSaveAs
VAR_INPUT
	i_bExecute					:BOOL;
	i_sSourcePath				:STRING;
	i_sDestinationPath			:STRING;
	i_sFileName					:STRING;
	i_sPrefix					:STRING;
END_VAR
VAR_OUTPUT
	q_bBusy						:BOOL;
	q_bDone						:BOOL;
	q_bError					:BOOL;
	q_sError					:STRING;
END_VAR
VAR
	fbSourceOpen				:FB_FileOpen;
	fbDestinationOpen			:FB_FileOpen;
	
	fbSourceRead				:FB_FileRead;
	fbDestinationWrite			:FB_FileWrite;
	
	fbSourceClose				:FB_FileClose;
	fbDestinationClose			:FB_FileClose;
	
	sSourceOpen					:STRING[300];
	sDestinationOpen			:STRING[300];

	arrData					:ARRAY[0..9999] OF BYTE;
	
	bOpen						:BOOL;
	bRead						:BOOL;
	bWrite						:BOOL;
	bClose						:BOOL;
	
	iStep						:INT;
END_VAR


CASE iStep OF
	
	0:
		q_bBusy:=FALSE;
		IF i_bExecute THEN
			q_sError:='';
			q_bError:=FALSE;
			q_bDone:=FALSE;
			q_bBusy:=TRUE;
			iStep:=10;
		END_IF

	10:
		sSourceOpen := CONCAT(i_sSourcePath,i_sFileName);
		sDestinationOpen := CONCAT(i_sDestinationPath,i_sPrefix);
		sDestinationOpen := CONCAT(sDestinationOpen,'_');
		sDestinationOpen := CONCAT(sDestinationOpen,i_sFileName);
		iStep:=20;
		
	20:
		bOpen:=TRUE;
		IF NOT fbSourceOpen.bBusy AND NOT fbDestinationOpen.bBusy AND NOT fbSourceOpen.bError AND NOT fbDestinationOpen.bError THEN
			iStep:=30;
		ELSIF fbSourceOpen.bError OR fbDestinationOpen.bError THEN
			q_bError:=TRUE;
			q_sError:='Error opening files';
			iStep:=50;
		END_IF
		
	30:
		bRead:=TRUE;
		IF fbSourceRead.bBusy THEN
			iStep:=35;
		END_IF
	35:
		
		IF NOT fbSourceRead.bBusy AND NOT fbSourceRead.bError THEN
			iStep:=40;
		ELSIF fbSourceRead.bError THEN
			q_bError:=TRUE;
			q_sError:='Error reading source file';
			iStep:=50;
		END_IF
		
	40:
		bWrite:=TRUE;
		IF fbDestinationWrite.bBusy THEN
			iStep:=45;
		END_IF
	45:
		IF NOT fbDestinationWrite.bBusy AND NOT fbDestinationWrite.bError THEN
			iStep:=50;
		ELSIF fbDestinationWrite.bError THEN
			q_bError:=TRUE;
			q_sError:='Error writing source file';
			iStep:=50;
		END_IF
	50:
		bClose:=TRUE;
		IF NOT fbSourceClose.bBusy AND NOT fbDestinationClose.bBusy AND NOT fbSourceClose.bError AND NOT fbDestinationClose.bError THEN
			iStep:=100;
		ELSIF fbSourceClose.bError OR fbDestinationClose.bError THEN
			q_bError:=TRUE;
			q_sError:='Error closing files';
			iStep:=0;
		END_IF
		
	100:
		q_bDone:=TRUE;
		iStep:=0;
	
END_CASE

Cmd();

ACTION Cmd:
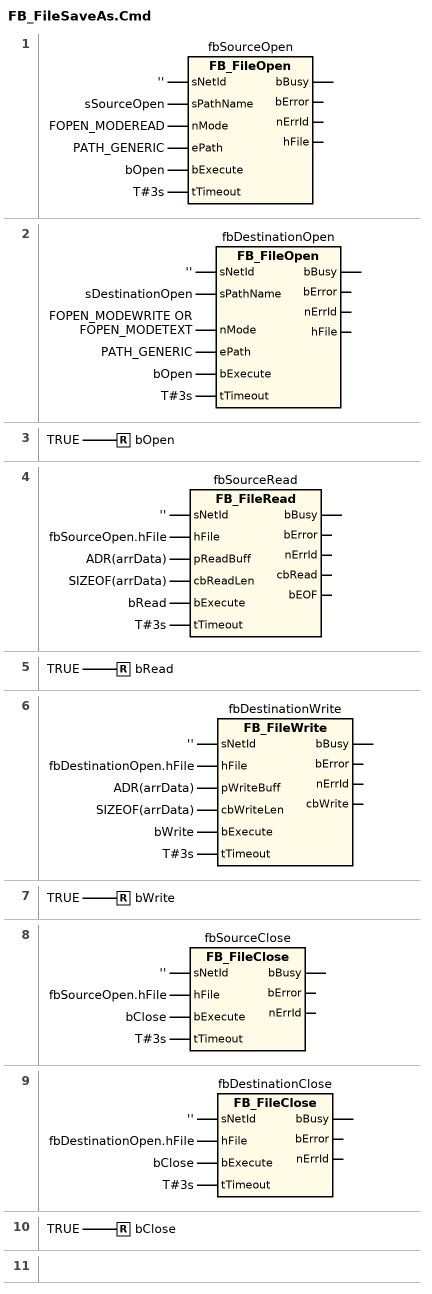
// NETWORK 1
fbSourceOpen(
    sNetId := '',
    sPathName := sSourceOpen,
    nMode := FOPEN_MODEREAD,
    ePath := PATH_GENERIC,
    bExecute := bOpen,
    tTimeout := T#3s); // FB_FileOpen

// NETWORK 2
fbDestinationOpen(
    sNetId := '',
    sPathName := sDestinationOpen,
    nMode := FOPEN_MODEWRITE OR FOPEN_MODETEXT,
    ePath := PATH_GENERIC,
    bExecute := bOpen,
    tTimeout := T#3s); // FB_FileOpen

// NETWORK 3
bOpen R= TRUE;

// NETWORK 4
fbSourceRead(
    sNetId := '',
    hFile := fbSourceOpen.hFile,
    pReadBuff := ADR(arrData),
    cbReadLen := SIZEOF(arrData),
    bExecute := bRead,
    tTimeout := T#3s); // FB_FileRead

// NETWORK 5
bRead R= TRUE;

// NETWORK 6
fbDestinationWrite(
    sNetId := '',
    hFile := fbDestinationOpen.hFile,
    pWriteBuff := ADR(arrData),
    cbWriteLen := SIZEOF(arrData),
    bExecute := bWrite,
    tTimeout := T#3s); // FB_FileWrite

// NETWORK 7
bWrite R= TRUE;

// NETWORK 8
fbSourceClose(sNetId := '', hFile := fbSourceOpen.hFile, bExecute := bClose, tTimeout := T#3s); // FB_FileClose

// NETWORK 9
fbDestinationClose(sNetId := '', hFile := fbDestinationOpen.hFile, bExecute := bClose, tTimeout := T#3s); // FB_FileClose

// NETWORK 10
bClose R= TRUE;

// NETWORK 11
END_ACTION

END_FUNCTION_BLOCK

// ---- POUs/3. Report/P3_07_SendReport.TcPOU
PROGRAM P3_07_SendReport
VAR
	fbSend				:FB_PythonScript;
	
	iError				:INT;
	tonResetError		:TON;
	
	iStep				:INT;
END_VAR

VAR PERSISTENT
	
END_VAR

tonResetError(IN:=(iError<>0),PT:=T#3S);
IF tonResetError.Q THEN
	iError:=0;
END_IF
CASE iStep OF
	
	0:
		IF GV.stReport.bStartSend_Sequence THEN
			GV.stReport.bStartSend_Sequence:=FALSE;
			iError:=0;
			iStep:=10;
		END_IF
	
	10:
		GV.stReport.bSend_Report:=TRUE;
		IF fbSend.q_bBusy THEN
			iStep:=15;
		END_IF
	
	15:
		IF NOT fbSend.q_bBusy AND fbSend.q_bDone THEN
			iStep:=999;
		ELSIF fbSend.q_bError THEN
			iError:=iStep;
			iStep:=999;
		END_IF
	
	999:
		iStep:=0;
END_CASE
ACT_CMDs();

ACTION ACT_CMDs:
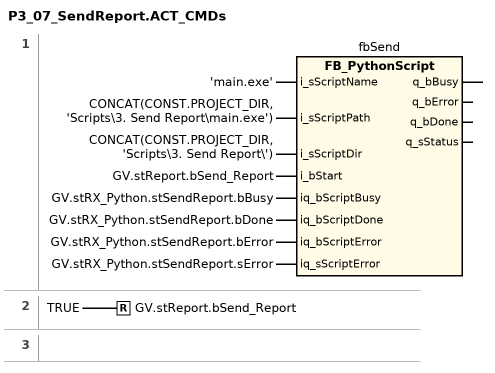
// NETWORK 1
fbSend(
    i_sScriptName := 'main.exe',
    i_sScriptPath := CONCAT(CONST.PROJECT_DIR,'Scripts\3. Send Report\main.exe'),
    i_sScriptDir := CONCAT(CONST.PROJECT_DIR,'Scripts\3. Send Report\'),
    i_bStart := GV.stReport.bSend_Report,
    iq_bScriptBusy := GV.stRX_Python.stSendReport.bBusy,
    iq_bScriptDone := GV.stRX_Python.stSendReport.bDone,
    iq_bScriptError := GV.stRX_Python.stSendReport.bError,
    iq_sScriptError := GV.stRX_Python.stSendReport.sError); // FB_PythonScript

// NETWORK 2
GV.stReport.bSend_Report R= TRUE;

// NETWORK 3
END_ACTION

END_PROGRAM

// ---- POUs/1. Main Control/P1_04_MachineControl.TcPOU
PROGRAM P1_04_MachineControl
VAR
	tonStarting		:TON;
	tonStopping		:TON;
	
	
	
	
	doorunlocked: INT;
	tofDoorLocked: TOF;
END_VAR

VAR PERSISTENT
	bBatchConfirmation1			:BOOL;
	bBatchConfirmation2			:BOOL;
	bBatchConfirmation3			:BOOL;
	bBatchConfirmation4			:BOOL;
END_VAR
VAR // added by the converter: edge detectors and wires of the graphical bodies
    _w1, _w2, _w3, _w4, _w5, _w6, _w7, _w8 : BOOL;
    _ft1 : F_TRIG;
    _rt1, _rt2 : R_TRIG;
END_VAR

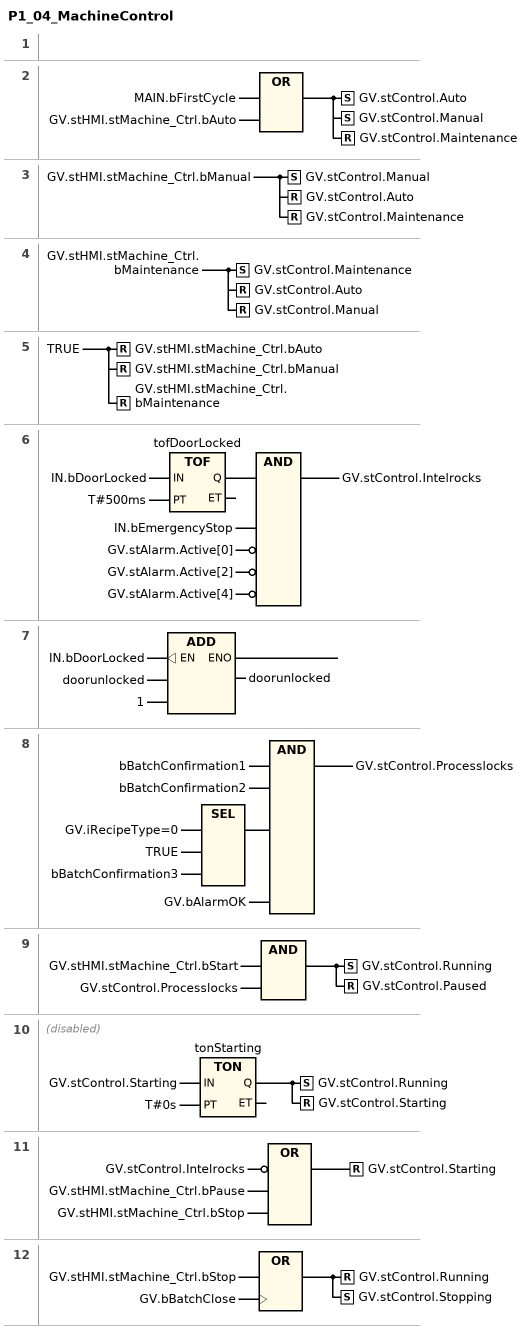
// NETWORK 1

// NETWORK 2
_w1 := MAIN.bFirstCycle OR GV.stHMI.stMachine_Ctrl.bAuto;
GV.stControl.Auto S= _w1;
GV.stControl.Manual S= _w1;
GV.stControl.Maintenance R= _w1;

// NETWORK 3
_w2 := GV.stHMI.stMachine_Ctrl.bManual;
GV.stControl.Manual S= _w2;
GV.stControl.Auto R= _w2;
GV.stControl.Maintenance R= _w2;

// NETWORK 4
_w3 := GV.stHMI.stMachine_Ctrl.bMaintenance;
GV.stControl.Maintenance S= _w3;
GV.stControl.Auto R= _w3;
GV.stControl.Manual R= _w3;

// NETWORK 5
GV.stHMI.stMachine_Ctrl.bAuto R= TRUE;
GV.stHMI.stMachine_Ctrl.bManual R= TRUE;
GV.stHMI.stMachine_Ctrl.bMaintenance R= TRUE;

// NETWORK 6
tofDoorLocked(IN := IN.bDoorLocked, PT := T#500ms); // TOF
GV.stControl.Intelrocks := tofDoorLocked.Q AND IN.bEmergencyStop AND NOT GV.stAlarm.Active[0] AND NOT GV.stAlarm.Active[2] AND NOT GV.stAlarm.Active[4];

// NETWORK 7
_ft1(CLK := IN.bDoorLocked);
IF _ft1.Q THEN doorunlocked := doorunlocked + 1; END_IF

// NETWORK 8
GV.stControl.Processlocks := bBatchConfirmation1 AND bBatchConfirmation2 AND SEL(GV.iRecipeType=0, TRUE, bBatchConfirmation3) AND GV.bAlarmOK;

// NETWORK 9
_w4 := GV.stHMI.stMachine_Ctrl.bStart AND GV.stControl.Processlocks;
GV.stControl.Running S= _w4;
GV.stControl.Paused R= _w4;

// NETWORK 10 (disabled)
// tonStarting(IN := GV.stControl.Starting, PT := T#0s); // TON
// GV.stControl.Running S= tonStarting.Q;
// GV.stControl.Starting R= tonStarting.Q;

// NETWORK 11
GV.stControl.Starting R= NOT GV.stControl.Intelrocks OR GV.stHMI.stMachine_Ctrl.bPause OR GV.stHMI.stMachine_Ctrl.bStop;

// NETWORK 12
_rt1(CLK := GV.bBatchClose);
_w5 := GV.stHMI.stMachine_Ctrl.bStop OR _rt1.Q;
GV.stControl.Running R= _w5;
GV.stControl.Stopping S= _w5;

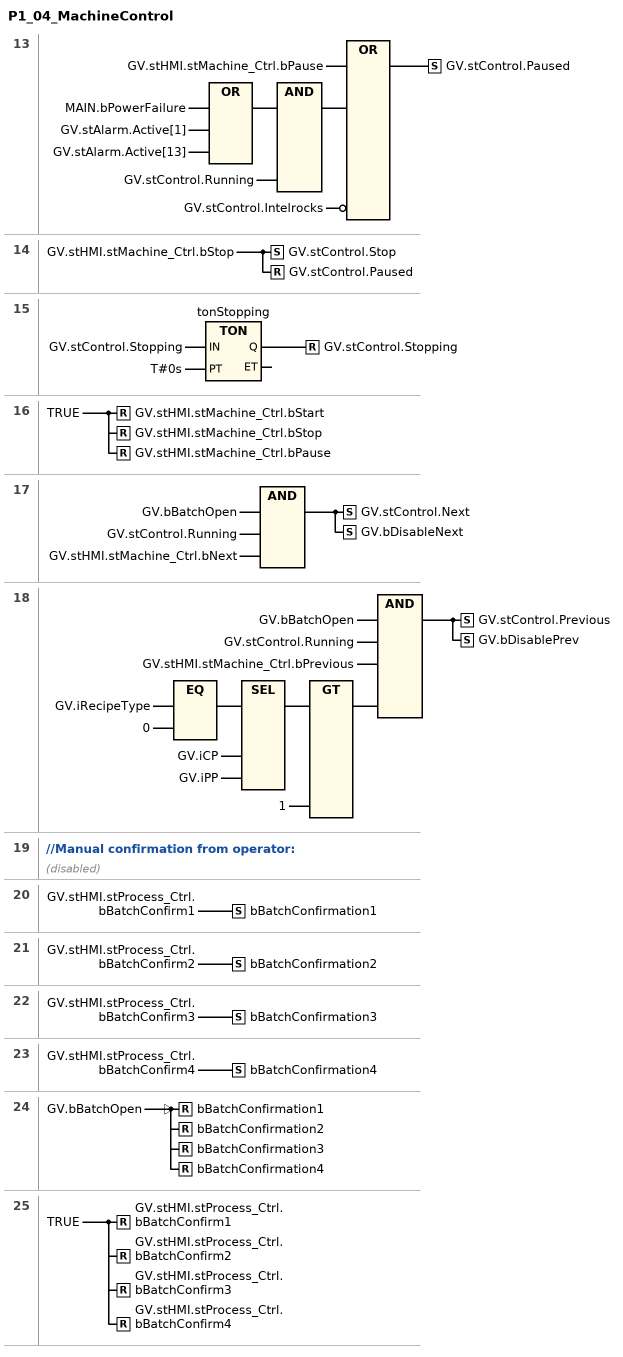
// NETWORK 13
GV.stControl.Paused S= GV.stHMI.stMachine_Ctrl.bPause OR (MAIN.bPowerFailure OR GV.stAlarm.Active[1] OR GV.stAlarm.Active[13]) AND GV.stControl.Running OR NOT GV.stControl.Intelrocks;

// NETWORK 14
_w6 := GV.stHMI.stMachine_Ctrl.bStop;
GV.stControl.Stop S= _w6;
GV.stControl.Paused R= _w6;

// NETWORK 15
tonStopping(IN := GV.stControl.Stopping, PT := T#0s); // TON
GV.stControl.Stopping R= tonStopping.Q;

// NETWORK 16
GV.stHMI.stMachine_Ctrl.bStart R= TRUE;
GV.stHMI.stMachine_Ctrl.bStop R= TRUE;
GV.stHMI.stMachine_Ctrl.bPause R= TRUE;

// NETWORK 17
_w7 := GV.bBatchOpen AND GV.stControl.Running AND GV.stHMI.stMachine_Ctrl.bNext;
GV.stControl.Next S= _w7;
GV.bDisableNext S= _w7;

// NETWORK 18
_w8 := GV.bBatchOpen AND GV.stControl.Running AND GV.stHMI.stMachine_Ctrl.bPrevious AND SEL(GV.iRecipeType = 0, GV.iCP, GV.iPP) > 1;
GV.stControl.Previous S= _w8;
GV.bDisablePrev S= _w8;

// NETWORK 19 (disabled)
// label: //Manual confirmation from operator

// NETWORK 20
bBatchConfirmation1 S= GV.stHMI.stProcess_Ctrl.bBatchConfirm1;

// NETWORK 21
bBatchConfirmation2 S= GV.stHMI.stProcess_Ctrl.bBatchConfirm2;

// NETWORK 22
bBatchConfirmation3 S= GV.stHMI.stProcess_Ctrl.bBatchConfirm3;

// NETWORK 23
bBatchConfirmation4 S= GV.stHMI.stProcess_Ctrl.bBatchConfirm4;

// NETWORK 24
_rt2(CLK := GV.bBatchOpen);
bBatchConfirmation1 R= _rt2.Q;
bBatchConfirmation2 R= _rt2.Q;
bBatchConfirmation3 R= _rt2.Q;
bBatchConfirmation4 R= _rt2.Q;

// NETWORK 25
GV.stHMI.stProcess_Ctrl.bBatchConfirm1 R= TRUE;
GV.stHMI.stProcess_Ctrl.bBatchConfirm2 R= TRUE;
GV.stHMI.stProcess_Ctrl.bBatchConfirm3 R= TRUE;
GV.stHMI.stProcess_Ctrl.bBatchConfirm4 R= TRUE;

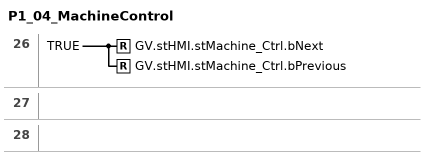
// NETWORK 26
GV.stHMI.stMachine_Ctrl.bNext R= TRUE;
GV.stHMI.stMachine_Ctrl.bPrevious R= TRUE;

// NETWORK 27

// NETWORK 28

END_PROGRAM

// ---- POUs/2. Process/P2_00_MAIN.TcPOU
PROGRAM P2_00_MAIN
VAR
	tonFlapReset			:TON;
END_VAR

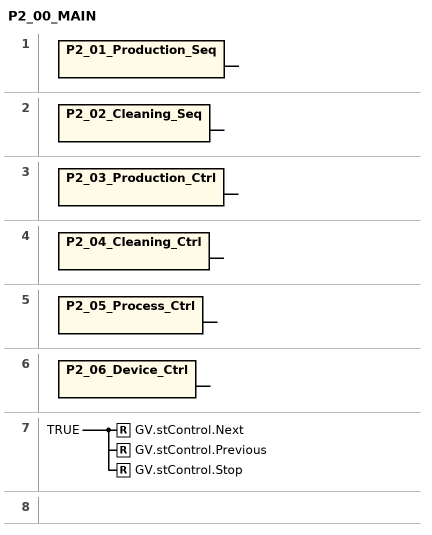
// NETWORK 1
P2_01_Production_Seq();

// NETWORK 2
P2_02_Cleaning_Seq();

// NETWORK 3
P2_03_Production_Ctrl();

// NETWORK 4
P2_04_Cleaning_Ctrl();

// NETWORK 5
P2_05_Process_Ctrl();

// NETWORK 6
P2_06_Device_Ctrl();

// NETWORK 7
GV.stControl.Next R= TRUE;
GV.stControl.Previous R= TRUE;
GV.stControl.Stop R= TRUE;

// NETWORK 8

END_PROGRAM

// ---- POUs/2. Process/P2_01_Production_Seq.TcPOU
PROGRAM P2_01_Production_Seq
VAR
	tDuration_TON				:ARRAY[0..10] OF TON;
	tDuration					:ARRAY[0..10] OF TIME;
	bRunning					:BOOL;
	
	trigStart					:R_TRIG;
	trigSkip					:R_TRIG;
	trigPrev					:R_TRIG;
	trigJump					:R_TRIG;
	
	iCountTotalProcess			:INT;
	iNoProceses					:INT;
	tTotalTime					:TON;
	trigResetTotal				:R_TRIG;
	
	bProcessRunning				:BOOL;
	bProcessFinish				:BOOL;

	iMaxNumberOfProcess			:INT;
	
	bPreviousStep				:BOOL;
END_VAR

VAR PERSISTENT
	bStartProcess				:BOOL;
	bStopProcess				:BOOL;
	
	iProcess					:INT;
	iStepPrev					:INT;
	iProcessPrev				:INT;
	iStep						:INT;
END_VAR

iMaxNumberOfProcess:=20;

GV.iPP:=iProcess;
IF iProcess > 1 THEN
	GV.iPrevPP:=iProcess-1;
END_IF


// Terminate process
IF GV.stControl.Stop THEN
	iStep := 1000;
END_IF

//Jump requests
trigStart(CLK:=GV.stControl.Running AND GV.iRecipeType=0);
trigSkip(CLK:=GV.stControl.Next);
trigPrev(CLK:=GV.stControl.Previous);
trigJump(CLK:=GV.stControl.Jump);

IF trigPrev.Q THEN
	bPreviousStep:=TRUE;
END_IF

//0 - Feeding
//1 - Mixing
//2 - Discharging

//Protect iProcess of forcing online value
IF iProcess < 1 THEN
	iProcess := 1;
ELSIF iProcess > iMaxNumberOfProcess THEN
	iProcess := iMaxNumberOfProcess;
END_IF

IF Recipes.Production_Active.stPhase[iProcess].iType=0 THEN
	bProcessRunning:=_Feeding.q_bRunning;
	bProcessFinish:=_Feeding.q_bFinished;
ELSIF Recipes.Production_Active.stPhase[iProcess].iType=1 THEN
	bProcessRunning:=_Mixing.q_bRunning;
	bProcessFinish:=_Mixing.q_bFinished;
ELSIF Recipes.Production_Active.stPhase[iProcess].iType=2 THEN
	bProcessRunning:=_Discharging.q_bRunning;
	bProcessFinish:=_Discharging.q_bFinished;
END_IF


CASE iStep OF 
	0:	
		iProcess := 0;
		iProcessPrev := 0;
		IF trigStart.Q THEN
			iProcess:=0;
			iStep := 200;
		END_IF
		
		IF iStep <> 0 THEN
			iStepPrev := 0;
		END_IF
		
	//Wait for process start
	200:
		bPreviousStep:=FALSE;
		bStartProcess:=TRUE;
		IF bProcessRunning THEN
			iStep:=300;
		END_IF
		
		IF iStep <> 200 THEN
			iStepPrev := 200;
		END_IF
	//Process running	
	300:
		IF bProcessFinish THEN
			iStep:=400;
		//not neccessery to change state if not running - affect phase pause timers
		ELSIF NOT GV.stControl.Running AND FALSE THEN
			iStep:=500;
		END_IF
		
		IF iStep <> 300 THEN
			iStepPrev := 300;
		END_IF
	//Process finish
	400:
		bStartProcess:=FALSE;
		bStopProcess:=TRUE;
		IF NOT bProcessRunning THEN
			bStopProcess:=FALSE;
			IF iProcess > 0 AND iProcess < iMaxNumberOfProcess AND NOT bPreviousStep THEN
				IF Recipes.Production_Active.stPhase[iProcess+1].bEnable THEN
					iProcessPrev:=iProcess;
					iProcess:=iProcess+1;
					iStep:=200;
				ELSE
					iStep:=1000;
				END_IF
			ELSIF bPreviousStep THEN
				iProcessPrev:=iProcess;
				IProcess:=iProcess-1;
				iStep:=200;
			END_IF
		END_IF
		
		IF iStep <> 400 THEN
			iStepPrev := 400;
		END_IF
	500:
		bStartProcess:=FALSE;
		IF GV.stControl.Running THEN
			iStep := 200;
		END_IF
	1000:
		bStartProcess:=FALSE;
		GV.stControl.Finish := TRUE;
		iStep := 0;
END_CASE

END_PROGRAM

// ---- POUs/2. Process/Production/_Feeding.TcPOU
PROGRAM _Feeding
VAR_INPUT
	i_bStart							:BOOL;
	i_bProcessFinished					:BOOL;
	i_bStepFinished						:BOOL;
	i_bSkipStep							:BOOL;
	i_bDischargeOpen					:BOOL;
	i_bDischargeClose					:BOOL;
	i_bEnableMixer						:BOOL;
	i_iMixer							:INT;
	i_rMixerSpeed						:REAL;	
END_VAR
VAR
	iStep								:INT;
	iPrevStep							:INT;
	Seq_TON								:ARRAY[0..9] OF TON;
	Seq_Time							:ARRAY[0..9] OF TIME;
	tonStepTime							:TON;
	bEnableMixer						:BOOL;
	trigEnableMixer						:R_TRIG;
END_VAR
VAR_OUTPUT
	q_bRunning						:BOOL;
	q_bFinished						:BOOL;
	q_stCmd							:ST_ProcessCmd;
	q_bDisCloseReq					:BOOL;
	q_tStepTime						:TIME;
END_VAR

q_bRunning:=iStep<>0;

IF i_bSkipStep THEN
	iStep:=1000;
END_IF

IF NOT i_bStart THEN
	iStep:=0;
END_IF

CASE iStep OF
	0:
		IF i_bStart THEN
			q_bFinished:=FALSE;
			iStep:=50;
		END_IF
		
		IF iStep <> 0 THEN
			iPrevStep:=0;
		END_IF
	
	50:
		IF i_bDischargeClose THEN
			iStep:=100;
		END_IF
		
		IF iStep <> 50 THEN
			iPrevStep:=50;
		END_IF
	
	100:
		
		IF i_bProcessFinished THEN
			iStep:=1000;
		END_IF
		IF iStep <> 100 THEN
			iPrevStep:=100;
		END_IF

		
	1000:
		q_bFinished:=TRUE;
		IF i_bStepFinished THEN
			iStep:=0;
		END_IF
END_CASE


q_bDisCloseReq:=F_StepCMP(iStep,50,0,0,0,0,0,0,0,0,0);

IF F_StepCMP(iStep,50,0,0,0,0,0,0,0,0,0) THEN
	q_stCmd.bDischargeOpen:=FALSE;
	q_stCmd.bDischargeClose:=TRUE;
ELSE
	q_stCmd.bDischargeOpen:=FALSE;
	q_stCmd.bDischargeClose:=FALSE;
END_IF

IF i_bEnableMixer THEN
	bEnableMixer:=NOT bEnableMixer;
END_IF

trigEnableMixer(CLK:=F_StepCMP(iStep,100,0,0,0,0,0,0,0,0,0));
IF trigEnableMixer.Q THEN
	bEnableMixer:=TRUE;
END_IF

IF F_StepCMP(iStep,100,0,0,0,0,0,0,0,0,0) AND bEnableMixer THEN
	q_stCmd.iMixer:=i_iMixer;
	q_stCmd.rMixerSpeed:=i_rMixerSpeed;
ELSE
	q_stCmd.iMixer:=0;
	q_stCmd.rMixerSpeed:=0;
	bEnableMixer:=FALSE;
END_IF

q_stCmd.bTightAir:=F_StepCMP(iStep,50,100,0,0,0,0,0,0,0,0) AND q_stCmd.iMixer <> 0;
q_stCmd.bChopper1_Air:=F_StepCMP(iStep,0,0,0,0,0,0,0,0,0,0) ;
q_stCmd.bChopper2_Air:=F_StepCMP(iStep,0,0,0,0,0,0,0,0,0,0);

//Statistic and Status
tonStepTime(IN:=q_bRunning,PT:=T#5H);
q_tStepTime:=tonStepTime.ET;

END_PROGRAM

// ---- POUs/2. Process/Production/_Mixing.TcPOU
PROGRAM _Mixing
VAR_INPUT
	i_bStart					:BOOL;
	i_bProcessFinished			:BOOL;
	i_bPause					:BOOL;
	i_bStepFinished				:BOOL;
	i_bSkipStep					:BOOL;
	i_bDischargeClose			:BOOL;
	i_iEndPoint					:INT;
	i_iMixer					:INT;
	i_rMixerSpeed				:REAL;
	i_iChopper					:INT;
	i_iTimeStep1				:ST_HMI_Time;
END_VAR
VAR
	iStep						:INT;
	iPrevStep					:INT;

	Seq_Time					:ARRAY[0..9] OF TIME;
	tonStepTime					:TON;
	
END_VAR
VAR_OUTPUT
	q_bRunning					:BOOL;
	q_bFinished					:BOOL;
	q_bDisCloseReq				:BOOL;
	q_stCmd						:ST_ProcessCmd;
	q_Seq_TON					:ARRAY[0..9] OF FB_TONP;
	q_tStepTime					:TIME;
END_VAR

//Recipe Parameters
Seq_Time[1]:=DINT_TO_TIME(i_iTimeStep1.mins)*60000 + 
			 DINT_TO_TIME(i_iTimeStep1.sec)*1000;			 
q_Seq_TON[1](IN:=iStep=100 OR GV.stControl.Paused,PAUSE:=GV.stControl.Paused,PT:=Seq_Time[1]);

q_bRunning:=iStep<>0;

IF i_bSkipStep THEN
	iStep:=1000;
END_IF

IF NOT i_bStart AND NOT GV.stControl.Paused THEN
	iStep:=0;
END_IF

CASE iStep OF
	0:
		IF i_bStart THEN
			q_bFinished:=FALSE;
			iStep:=50;
		END_IF
		
		IF iStep <> 0 THEN
			iPrevStep:=0;
		END_IF
	50:
		IF i_bDischargeClose THEN
			iStep:=100;
		END_IF
		
		IF iStep <> 50 THEN
			iPrevStep:=50;
		END_IF
	
	//Mixing
	100:
		IF (q_Seq_TON[1].Q AND i_iEndPoint=0) OR (i_bProcessFinished AND i_iEndpoint=1) THEN
			iStep:=1000;
		END_IF
		IF iStep <> 100 THEN
			iPrevStep:=100;
		END_IF
		
	1000:
		q_bFinished:=TRUE;
		IF i_bStepFinished THEN
			iStep:=0;
		END_IF
END_CASE


q_bDisCloseReq:=F_StepCMP(iStep,50,0,0,0,0,0,0,0,0,0);

IF F_StepCMP(iStep,50,0,0,0,0,0,0,0,0,0) THEN
	q_stCmd.bDischargeOpen:=FALSE;
	q_stCmd.bDischargeClose:=TRUE;
ELSE
	q_stCmd.bDischargeOpen:=FALSE;
	q_stCmd.bDischargeClose:=FALSE;
END_IF

IF F_StepCMP(iStep,100,0,0,0,0,0,0,0,0,0) AND NOT i_bPause THEN
	q_stCmd.iMixer:=i_iMixer;
	q_stCmd.rMixerSpeed:=i_rMixerSpeed;
ELSE
	q_stCmd.iMixer:=0;
	q_stCmd.rMixerSpeed:=0;
END_IF

IF F_StepCMP(iStep,100,0,0,0,0,0,0,0,0,0) AND NOT i_bPause THEN
	q_stCmd.iChopper:=i_iChopper;
ELSE
	q_stCmd.iChopper:=0;
END_IF

q_stCmd.bTightAir:=F_StepCMP(iStep,100,0,0,0,0,0,0,0,0,0);
q_stCmd.bChopper1_Air:=F_StepCMP(iStep,100,0,0,0,0,0,0,0,0,0);
q_stCmd.bChopper2_Air:=F_StepCMP(iStep,100,0,0,0,0,0,0,0,0,0);

//Statistic and Status
tonStepTime(IN:=q_bRunning,PT:=T#5H);
q_tStepTime:=tonStepTime.ET;

END_PROGRAM

// ---- FB/FB_TONP.TcPOU
FUNCTION_BLOCK FB_TONP
VAR_INPUT
	IN				:BOOL;
	PAUSE			:BOOL;
	PT				:TIME;
END_VAR
	
VAR_OUTPUT
	ET				:TIME;
	Q				:BOOL;
END_VAR
VAR
	TON				:TON;
	trigPause		:R_TRIG;
	trigStart		:R_TRIG;
	PT_START		:TIME;
	ET_PAUSE		:TIME;
END_VAR

trigStart(CLK:=IN);
trigPause(CLK:=PAUSE);

PT_START:=PT;
IF trigStart.Q THEN
	ET_PAUSE:=T#0S;
END_IF
IF IN AND trigPause.Q THEN
	ET_PAUSE:=TON.ET + ET_PAUSE;
END_IF


TON(IN:=IN AND NOT PAUSE ,PT:=SEL(TO_DINT(PT_START)-TO_DINT(ET_PAUSE)>0,T#0S,PT_START-ET_PAUSE));

Q:=TON.Q;
ET:=(ET_PAUSE+TON.ET);
IF NOT IN THEN
	ET:=T#0s;
END_IF

END_FUNCTION_BLOCK

// ---- POUs/2. Process/P2_02_Cleaning_Seq.TcPOU
PROGRAM P2_02_Cleaning_Seq
VAR
	tDuration_TON				:ARRAY[0..10] OF TON;
	tDuration					:ARRAY[0..10] OF TIME;
	bRunning					:BOOL;
	
	trigStart					:R_TRIG;
	trigSkip					:R_TRIG;
	trigPrev					:R_TRIG;
	trigJump					:R_TRIG;
	
	iCountTotalProcess			:INT;
	iNoProceses					:INT;
	tTotalTime					:TON;
	trigResetTotal				:R_TRIG;
	
	bProcessRunning				:BOOL;
	bProcessFinish				:BOOL;
	
	iMaxNumberOfProcess			:INT;
	bPreviousStep				:BOOL;
END_VAR

VAR PERSISTENT
	bStartProcess				:BOOL;
	bStopProcess				:BOOL;
	
	iProcess					:INT;
	iStepPrev					:INT;
	iProcessPrev				:INT;
	iStep						:INT;
END_VAR

iMaxNumberOfProcess:=20;

GV.iCP:=iProcess;
IF iProcess > 1 THEN
	GV.iPrevCP:=iProcess-1;
END_IF


// Terminate process
IF GV.stControl.Stop THEN
	iStep := 1000;
END_IF

//Jump requests
trigStart(CLK:=GV.stControl.Running AND GV.iRecipeType=1);
trigSkip(CLK:=GV.stControl.Next);
trigPrev(CLK:=GV.stControl.Previous);
trigJump(CLK:=GV.stControl.Jump);

IF trigPrev.Q THEN
	bPreviousStep:=TRUE;
END_IF

//0 - Feeding
//1 - Mixing
//2 - Discharging

//Protect iProcess of forcing online value
IF iProcess < 0 THEN
	iProcess := 0;
ELSIF iProcess > iMaxNumberOfProcess THEN
	iProcess := iMaxNumberOfProcess;
END_IF

IF Recipes.Cleaning_Active.stPhase[iProcess].iType = 0 THEN
	bProcessRunning:=_PreWash.q_bRunning;
	bProcessFinish:=_PreWash.q_bFinished;
ELSIF Recipes.Cleaning_Active.stPhase[iProcess].iType = 1 THEN
	bProcessRunning:=_Mounting.q_bRunning;
	bProcessFinish:=_Mounting.q_bFinished;
ELSIF Recipes.Cleaning_Active.stPhase[iProcess].iType = 2 THEN
	bProcessRunning:=_MainClean.q_bRunning;
	bProcessFinish:=_MainClean.q_bFinished;
ELSIF Recipes.Cleaning_Active.stPhase[iProcess].iType = 3 THEN
	bProcessRunning:=FALSE;
	bProcessFinish:=FALSE;
ELSIF Recipes.Cleaning_Active.stPhase[iProcess].iType = 4 THEN
	bProcessRunning:=_Draining.q_bRunning;
	bProcessFinish:=_Draining.q_bFinished;
ELSIF Recipes.Cleaning_Active.stPhase[iProcess].iType = 5 THEN
	bProcessRunning:=_Blowing.q_bRunning;
	bProcessFinish:=_Blowing.q_bFinished;
ELSIF Recipes.Cleaning_Active.stPhase[iProcess].iType = 6 THEN
	bProcessRunning:=_Control.q_bRunning;
	bProcessFinish:=_Control.q_bFinished;
END_IF


CASE iStep OF 
	0:	
		iProcess := 0;
		iProcessPrev := 0;
		IF trigStart.Q THEN
			iProcess:=1;
			iStep := 200;
		END_IF
		
		IF iStep <> 0 THEN
			iStepPrev := 0;
		END_IF

		
	//Wait for process start
	200:
		bPreviousStep:=FALSE;
		bStartProcess:=TRUE;
		IF bProcessRunning THEN
			iStep:=300;
		END_IF
		
		IF iStep <> 200 THEN
			iStepPrev := 200;
		END_IF
	//Process running	
	300:
		IF bProcessFinish THEN
			iStep:=400;
		END_IF
		
		IF iStep <> 300 THEN
			iStepPrev := 300;
		END_IF
	//Process finish
	400:
		bStartProcess:=FALSE;
		bStopProcess:=TRUE;
		IF NOT bProcessRunning THEN
			bStopProcess:=FALSE;
			IF iProcess > 0 AND iProcess < iMaxNumberOfProcess AND NOT bPreviousStep THEN
				IF Recipes.Cleaning_Active.stPhase[iProcess+1].bEnable THEN
					iProcessPrev:=iProcess;
					iProcess:=iProcess+1;
					iStep:=200;
				ELSE
					iStep:=1000;
				END_IF
			ELSIF bPreviousStep THEN
				iProcessPrev:=iProcess;
				IProcess:=iProcess-1;
				iStep:=200;
			END_IF
		END_IF
		IF iStep <> 400 THEN
			iStepPrev := 400;
		END_IF
	500:
		bStartProcess:=FALSE;
		IF GV.stControl.Running THEN
			iStep := 200;
		END_IF
	1000:
		bStartProcess:=FALSE;
		GV.stControl.Finish := TRUE;
		iStep := 0;
END_CASE

END_PROGRAM

// ---- POUs/2. Process/Cleaning/_PreWash.TcPOU
PROGRAM _PreWash
VAR_INPUT
	i_bStart					:BOOL;
	i_bPause					:BOOL;
	i_bStepFinished				:BOOL;
	i_bSkipStep					:BOOL;
	i_bFlapMode					:BOOL;
	i_bDischargeOpened			:BOOL;
	i_bDischargeClosed			:BOOL;
	i_iMedium					:INT;
	i_iMixer					:INT;
	i_rMixerSpeed				:REAL;
	i_iChopper					:INT;
	i_iTimeStep1				:ST_HMI_Time;
END_VAR
VAR
	iStep						:INT;
	iPrevStep					:INT;
	Seq_Time					:ARRAY[0..9] OF TIME;
	tonStepTime					:TON;
END_VAR
VAR_OUTPUT
	q_bRunning					:BOOL;
	q_bFinished					:BOOL;
	q_stCmd						:ST_ProcessCmd;
	q_bDisOpenReq				:BOOL;
	q_tStepTime					:TIME;
	q_Seq_TON					:ARRAY[0..9] OF FB_TONP;
END_VAR

//Recipe Parameters
Seq_Time[1]:=DINT_TO_TIME(i_iTimeStep1.mins)*60000 + 
			 DINT_TO_TIME(i_iTimeStep1.sec)*1000;
		 
q_Seq_TON[1](IN:=iStep=100,PAUSE:=i_bPause,PT:=Seq_Time[1]);

q_bRunning:=iStep<>0;

IF i_bSkipStep THEN
	iStep:=1000;
END_IF

IF NOT i_bStart THEN
	iStep:=0;
END_IF

CASE iStep OF
	0:
		IF i_bStart THEN
			q_bFinished:=FALSE;
			iStep:=50;
		END_IF
		
		IF iStep <> 0 THEN
			iPrevStep:=0;
		END_IF
	
	//Wait for discharge flap to be opened
	50:
		IF i_bDischargeOpened THEN
			IF iPrevStep=0 THEN
				iStep:=100;
			ELSE
				iStep:=iPrevStep;
			END_IF
		END_IF
	
	//Cleaning time
	100:
		IF q_Seq_TON[1].Q THEN
			iStep:=1000;
		END_IF
		
		IF iStep <> 100 THEN
			iPrevStep:=100;
		END_IF
		
	1000:
		q_bFinished:=TRUE;
		IF i_bStepFinished THEN
			iStep:=0;
		END_IF
END_CASE

q_bDisOpenReq:=F_StepCMP(iStep,50,0,0,0,0,0,0,0,0,0);

IF F_StepCMP(iStep,50,0,0,0,0,0,0,0,0,0) THEN
	q_stCmd.bDischargeClose:=FALSE;
	q_stCmd.bDischargeOpen:=TRUE;
ELSE
	q_stCmd.bDischargeClose:=FALSE;
	q_stCmd.bDischargeOpen:=FALSE;
END_IF

IF F_StepCMP(iStep,100,0,0,0,0,0,0,0,0,0) AND NOT i_bPause THEN
	q_stCmd.iMixer:=i_iMixer;
	q_stCmd.rMixerSpeed:=i_rMixerSpeed;
ELSE
	q_stCmd.iMixer:=0;
	q_stCmd.rMixerSpeed:=0;
END_IF

IF F_StepCMP(iStep,100,0,0,0,0,0,0,0,0,0) AND NOT i_bPause THEN
	q_stCmd.iChopper:=i_iChopper;
ELSE
	q_stCmd.iChopper:=0;
END_IF

q_stCmd.bAir:=F_StepCMP(iStep,0,0,0,0,0,0,0,0,0,0);
q_stCmd.bWater:=F_StepCMP(iStep,100,0,0,0,0,0,0,0,0,0) AND ((i_iMedium = 0)OR(i_iMedium = 1));
q_stCmd.bColdWater:=F_StepCMP(iStep,100,0,0,0,0,0,0,0,0,0) AND (i_iMedium = 0);
q_stCmd.bWarmWater:=F_StepCMP(iStep,100,0,0,0,0,0,0,0,0,0) AND (i_iMedium = 1);
q_stCmd.bProcessWater:=F_StepCMP(iStep,100,0,0,0,0,0,0,0,0,0) AND (i_iMedium = 2);

q_stCmd.bTightAir:=F_StepCMP(iStep,50,100,0,0,0,0,0,0,0,0);

q_stCmd.bChopper1_Water:=F_StepCMP(iStep,100,0,0,0,0,0,0,0,0,0);
q_stCmd.bChopper2_Water:=F_StepCMP(iStep,100,0,0,0,0,0,0,0,0,0);

//Statistic and Status
tonStepTime(IN:=q_bRunning,PT:=T#5H);
q_tStepTime:=tonStepTime.ET;

END_PROGRAM

// ---- POUs/2. Process/Cleaning/_Mounting.TcPOU
PROGRAM _Mounting
VAR_INPUT
	i_bStart						:BOOL;
	i_bStepFinished					:BOOL;
	i_bProcessFinished				:BOOL;
	i_bSkipStep						:BOOL;
END_VAR
VAR
	iStep							:INT;
	tonStepTime						:TON;
END_VAR
VAR_OUTPUT
	q_bRunning						:BOOL;
	q_bFinished						:BOOL;
	q_stCmd							:ST_ProcessCmd;
	q_bReqFlapOpen					:BOOL;
	q_bReqFlapClosed				:BOOL;
	q_tStepTime						:TIME;
END_VAR

q_bRunning:=iStep<>0;

IF i_bSkipStep THEN
	iStep:=1000;
END_IF

IF NOT i_bStart THEN
	iStep:=0;
END_IF

CASE iStep OF
	0:
		IF i_bStart THEN
			q_bFinished:=FALSE;
			iStep:=50;
		END_IF
	
	//Mixer and Choppers are rotating
	50:
		IF i_bProcessFinished THEN
			iStep:=1000;
		END_IF
	
		
	1000:
		q_bFinished:=TRUE;
		IF i_bStepFinished THEN
			iStep:=0;
		END_IF
END_CASE


//Statistic and Status
tonStepTime(IN:=q_bRunning,PT:=T#5H);
q_tStepTime:=tonStepTime.ET;

END_PROGRAM

// ---- POUs/2. Process/Cleaning/_MainClean.TcPOU
PROGRAM _MainClean
VAR_INPUT
	i_bStart					:BOOL;
	i_bPause					:BOOL;
	i_bStepFinished				:BOOL;
	i_bSkipStep					:BOOL;
	i_bDischargeOpened			:BOOL;
	i_bDischargeClosed			:BOOL;
	i_iMedium					:INT;
	i_iDetergent				:INT;
	i_bDetergentConfirm			:BOOL;
	i_bDischargeConfirm			:BOOL;
	i_iMixer					:INT;
	i_rMixerSpeed				:REAL;
	i_iChopper					:INT;
	i_iTimeStep1				:ST_HMI_Time;
	i_iTimeStep2				:ST_HMI_Time;
	i_iTimeStep3				:ST_HMI_Time;

END_VAR
VAR
	iStep						:INT;
	iPrevStep					:INT;
	Seq_Time					:ARRAY[0..9] OF TIME;
	tonStepTime					:TON;
END_VAR
VAR_OUTPUT
	q_bRunning					:BOOL;
	q_bFinished					:BOOL;
	q_stCmd						:ST_ProcessCmd;
	q_bDetergentReq				:BOOL;
	q_bDisOpenReq				:BOOL;
	q_bDisCloseReq				:BOOL;
	q_bDischargeReq				:BOOL;
	q_tStepTime					:TIME;
	q_Seq_TON					:ARRAY[0..9] OF FB_TONP;
END_VAR

//Recipe Parameters
Seq_Time[1]:=DINT_TO_TIME(i_iTimeStep1.mins)*60000 + 
			 DINT_TO_TIME(i_iTimeStep1.sec)*1000;
Seq_Time[2]:=DINT_TO_TIME(i_iTimeStep2.mins)*60000 + 
			 DINT_TO_TIME(i_iTimeStep2.sec)*1000;
Seq_Time[3]:=DINT_TO_TIME(i_iTimeStep3.mins)*60000 + 
			 DINT_TO_TIME(i_iTimeStep3.sec)*1000;

			 
q_Seq_TON[1](IN:=iStep=100,PAUSE:=i_bPause,PT:=Seq_Time[1]);
q_Seq_TON[2](IN:=iStep=200,PAUSE:=i_bPause,PT:=Seq_Time[2]);
q_Seq_TON[3](IN:=iStep=300,PAUSE:=i_bPause,PT:=Seq_Time[3]);


q_bRunning:=iStep<>0;

IF i_bSkipStep THEN
	iStep:=1000;
END_IF

IF NOT i_bStart THEN
	iStep:=0;
END_IF

CASE iStep OF
	0:
		IF i_bStart THEN
			q_bFinished:=FALSE;
			iStep:=50;
		END_IF
		
		IF iStep <> 0 THEN
			iPrevStep:=0;
		END_IF
	
	//Wait for discharge flap top be closed
	50:
		IF i_bDischargeClosed THEN
			iStep:=100;
		END_IF
	
	//Filling time
	100:
		IF q_Seq_TON[1].Q THEN
			iStep:=150;
		END_IF
		
		IF iStep <> 100 THEN
			iPrevStep:=100;
		END_IF
	
	//Wait for detergent confirmation
	150:
		IF (i_iDetergent = 0) OR (i_iDetergent = 1 AND i_bDetergentConfirm) THEN
			iStep:=200;
		END_IF
		
		IF iStep <> 150 THEN
			iPrevStep:=150;	
		END_IF
		
	//Cleaning time
	200:
		IF q_Seq_TON[2].Q THEN
			iStep:=250;
		END_IF
		
		IF iStep <> 200 THEN
			iPrevStep:=200;
		END_IF
	
	//Wait for discharge flap to be opened	
	250:
		IF i_bDischargeOpened THEN
			iStep:=300;
		END_IF
		
	//Discharge time
	300:
		IF q_Seq_TON[3].Q OR GV.stSettings.bDischargeFlap_Manual THEN
			iStep:=350;
		END_IF	
		
		IF iStep <> 300 THEN
			iPrevStep:=300;
		END_IF
		
	//Confirmation that water is discharged
	350:
		IF (GV.stSettings.bDischargeFlap_Manual AND i_bDischargeConfirm) OR NOT GV.stSettings.bDischargeFlap_Manual THEN
			iStep:=400;
		END_IF
	
	400:
		IF i_bDischargeClosed THEN
			iStep:=1000;
		END_IF
	
	1000:
		q_bFinished:=TRUE;
		IF i_bStepFinished THEN
			iStep:=0;
		END_IF
END_CASE

q_bDisOpenReq:=F_StepCMP(iStep,250,0,0,0,0,0,0,0,0,0);
q_bDisCloseReq:=F_StepCMP(iStep,50,400,0,0,0,0,0,0,0,0);
q_bDischargeReq:=F_StepCMP(iStep,350,0,0,0,0,0,0,0,0,0);

IF F_StepCMP(iStep,50,400,0,0,0,0,0,0,0,0) THEN
	q_stCmd.bDischargeOpen:=FALSE;
	q_stCmd.bDischargeClose:=TRUE;
ELSIF F_StepCMP(iStep,250,0,0,0,0,0,0,0,0,0) THEN
	q_stCmd.bDischargeClose:=FALSE;
	q_stCmd.bDischargeOpen:=FALSE;
	q_stCmd.bDischargeHalfOpen:=TRUE;
ELSIF NOT F_StepCMP(iStep,250,0,0,0,0,0,0,0,0,0) AND NOT F_StepCMP(iStep,50,0,0,0,0,0,0,0,0,0) THEN
	q_stCmd.bDischargeClose:=FALSE;
	q_stCmd.bDischargeOpen:=FALSE;
	q_stCmd.bDischargeHalfOpen:=FALSE;
END_IF

IF F_StepCMP(iStep,100,200,0,0,0,0,0,0,0,0) AND NOT i_bPause THEN
	q_stCmd.iMixer:=i_iMixer;
	q_stCmd.rMixerSpeed:=i_rMixerSpeed;
ELSIF F_StepCMP(iStep,300,0,0,0,0,0,0,0,0,0) AND NOT i_bPause THEN
	q_stCmd.iMixer:=i_iMixer;
	q_stCmd.rMixerSpeed:=GV.stSettings.rMixerDischargeSpeed;
ELSE
	q_stCmd.iMixer:=0;
	q_stCmd.rMixerSpeed:=0;
END_IF

IF F_StepCMP(iStep,100,0,0,0,0,0,0,0,0,0) AND 
	TO_DINT(q_Seq_TON[1].ET)/60000 > GV.stSettings.iFillingChopperOnTime AND NOT i_bPause THEN
	q_stCmd.iChopper:=i_iChopper;
ELSIF F_StepCMP(iStep,200,0,0,0,0,0,0,0,0,0) AND NOT i_bPause THEN
	q_stCmd.iChopper:=i_iChopper;
ELSE
	q_stCmd.iChopper:=0;
END_IF

q_stCmd.bAir:=F_StepCMP(iStep,0,0,0,0,0,0,0,0,0,0);
q_stCmd.bWater:=F_StepCMP(iStep,100,0,0,0,0,0,0,0,0,0) AND ((i_iMedium = 0)OR(i_iMedium = 1));
q_stCmd.bColdWater:=F_StepCMP(iStep,100,0,0,0,0,0,0,0,0,0) AND (i_iMedium = 0);
q_stCmd.bWarmWater:=F_StepCMP(iStep,100,0,0,0,0,0,0,0,0,0) AND (i_iMedium = 1);
q_stCmd.bProcessWater:=F_StepCMP(iStep,100,0,0,0,0,0,0,0,0,0) AND (i_iMedium = 2);

q_stCmd.bTightAir:=F_StepCMP(iStep,50,100,150,200,300,0,0,0,0,0);
q_stCmd.bChopper1_Air:=F_StepCMP(iStep,50,150,200,300,0,0,0,0,0,0);
q_stCmd.bChopper2_Air:=F_StepCMP(iStep,50,150,200,300,0,0,0,0,0,0);


q_stCmd.bChopper1_Water:=F_StepCMP(iStep,100,0,0,0,0,0,0,0,0,0);
q_stCmd.bChopper2_Water:=F_StepCMP(iStep,100,0,0,0,0,0,0,0,0,0);

//Wait for requests
q_bDetergentReq:=F_StepCMP(iStep,150,0,0,0,0,0,0,0,0,0);

//Statistic and Status
tonStepTime(IN:=q_bRunning,PT:=T#5H);
q_tStepTime:=tonStepTime.ET;

END_PROGRAM

// ---- POUs/2. Process/Cleaning/_Draining.TcPOU
PROGRAM _Draining
VAR_INPUT
	i_bStart					:BOOL;
	i_bPause					:BOOL;
	i_bStepFinished				:BOOL;
	i_bSkipStep					:BOOL;
	i_bDischargeOpened			:BOOL;
	i_bDischargeClosed			:BOOL;
	i_iTimeStep1				:ST_HMI_Time;
END_VAR
VAR
	iStep						:INT;
	Seq_Time					:ARRAY[0..9] OF TIME;
	tonStepTime					:TON;
END_VAR
VAR_OUTPUT
	q_bRunning						:BOOL;
	q_bFinished						:BOOL;
	q_stCmd							:ST_ProcessCmd;
	q_bDisOpenReq					:BOOL;
	q_tStepTime						:TIME;
	q_Seq_TON						:ARRAY[0..9] OF FB_TONP;
END_VAR

//Recipe Parameters
Seq_Time[1]:=DINT_TO_TIME(i_iTimeStep1.mins)*60000 + 
			 DINT_TO_TIME(i_iTimeStep1.sec)*1000;
		 
q_Seq_TON[1](IN:=iStep=100,PAUSE:=i_bPause,PT:=Seq_Time[1]);

q_bRunning:=iStep<>0;

IF i_bSkipStep THEN
	iStep:=1000;
END_IF

IF NOT i_bStart THEN
	iStep:=0;
END_IF

CASE iStep OF
	0:
		IF i_bStart THEN
			q_bFinished:=FALSE;
			iStep:=50;
		END_IF
	
	//Mixer and Choppers are rotating
	50:
		IF i_bDischargeOpened THEN
			iStep:=100;
		END_IF
	
	//Draining
	100:
		IF q_Seq_TON[1].Q THEN
			iStep:=1000;
		END_IF
		
	1000:
		q_bFinished:=TRUE;
		IF i_bStepFinished THEN
			iStep:=0;
		END_IF
END_CASE


q_stCmd.iMixer:=0;
q_stCmd.rMixerSpeed:=0;
q_stCmd.iChopper:=0;

q_bDisOpenReq:=F_StepCMP(iStep,50,0,0,0,0,0,0,0,0,0);

IF F_StepCMP(iStep,50,0,0,0,0,0,0,0,0,0) THEN
	q_stCmd.bDischargeClose:=FALSE;
	q_stCmd.bDischargeOpen:=TRUE;
ELSE
	q_stCmd.bDischargeClose:=FALSE;
	q_stCmd.bDischargeOpen:=FALSE;
END_IF

q_stCmd.bChopper1_Water:=F_StepCMP(iStep,100,0,0,0,0,0,0,0,0,0);
q_stCmd.bChopper2_Water:=F_StepCMP(iStep,100,0,0,0,0,0,0,0,0,0);
q_stCmd.bChopper1_Drain:=F_StepCMP(iStep,100,0,0,0,0,0,0,0,0,0);
q_stCmd.bChopper2_Drain:=F_StepCMP(iStep,100,0,0,0,0,0,0,0,0,0);

//Statistic and Status
tonStepTime(IN:=q_bRunning,PT:=T#5H);
q_tStepTime:=tonStepTime.ET;

END_PROGRAM

// ---- POUs/2. Process/Cleaning/_Blowing.TcPOU
PROGRAM _Blowing
VAR_INPUT
	i_bStart							:BOOL;
	i_bPause							:BOOL;
	i_bStepFinished						:BOOL;
	i_bSkipStep							:BOOL;
	i_bDischargeOpened					:BOOL;
	i_bDischargeClosed					:BOOL;
	i_iMixer							:INT;
	i_rMixerSpeed						:REAL;
	i_iChopper							:INT;
	i_iTimeStep1						:ST_HMI_Time; 		
END_VAR
VAR
	iStep						:INT;
	iPrevStep					:INT;
	Seq_Time					:ARRAY[0..9] OF TIME;
	tonStepTime					:TON;
END_VAR
VAR_OUTPUT
	q_bRunning						:BOOL;
	q_bFinished						:BOOL;
	q_stCmd							:ST_ProcessCmd;
	q_bDisOpenReq					:BOOL;
	q_tStepTime						:TIME;
	q_Seq_TON						:ARRAY[0..9] OF FB_TONP;
END_VAR

//Recipe Parameters
Seq_Time[1]:=DINT_TO_TIME(i_iTimeStep1.mins)*60000 + 
			 DINT_TO_TIME(i_iTimeStep1.sec)*1000;

		 
q_Seq_TON[1](IN:=iStep=100,PAUSE:=i_bPause,PT:=Seq_Time[1]);

q_bRunning:=iStep<>0;

IF i_bSkipStep THEN
	iStep:=1000;
END_IF

IF NOT i_bStart THEN
	iStep:=0;
END_IF

CASE iStep OF
	0:
		IF i_bStart THEN
			q_bFinished:=FALSE;
			iStep:=50;
		END_IF
		
		IF iStep <> 0 THEN
			iPrevStep:=0;
		END_IF
	
	//Wait for open discharge valve to be open
	50:
		IF i_bDischargeOpened THEN
			iStep:=100;
		END_IF
		IF iStep <> 50 THEN
			iPrevStep:=50;
		END_IF
	
	//Blowing time filter housing
	100:
		IF q_Seq_TON[1].Q THEN
			iStep:=1000;
		END_IF
		
		IF iStep <> 100 THEN
			iPrevStep:=100;
		END_IF
	1000:
		q_bFinished:=TRUE;
		IF i_bStepFinished THEN
			iStep:=0;
		END_IF
END_CASE

q_bDisOpenReq:=F_StepCMP(iStep,50,0,0,0,0,0,0,0,0,0);

IF F_StepCMP(iStep,50,0,0,0,0,0,0,0,0,0) THEN
	q_stCmd.bDischargeClose:=FALSE;
	q_stCmd.bDischargeOpen:=TRUE;
ELSE
	q_stCmd.bDischargeClose:=FALSE;
	q_stCmd.bDischargeOpen:=FALSE;
END_IF

IF F_StepCMP(iStep,100,0,0,0,0,0,0,0,0,0) AND NOT i_bPause THEN
	q_stCmd.iMixer:=i_iMixer;
	q_stCmd.rMixerSpeed:=i_rMixerSpeed;
ELSE
	q_stCmd.iMixer:=0;
	q_stCmd.rMixerSpeed:=0;
END_IF

IF F_StepCMP(iStep,100,0,0,0,0,0,0,0,0,0) AND NOT i_bPause THEN
	q_stCmd.iChopper:=i_iChopper;
ELSE
	q_stCmd.iChopper:=0;
END_IF

q_stCmd.bAir:=F_StepCMP(iStep,100,0,0,0,0,0,0,0,0,0);
q_stCmd.bWater:=F_StepCMP(iStep,0,0,0,0,0,0,0,0,0,0);
q_stCmd.bColdWater:=F_StepCMP(iStep,0,0,0,0,0,0,0,0,0,0);
q_stCmd.bWarmWater:=F_StepCMP(iStep,0,0,0,0,0,0,0,0,0,0);
q_stCmd.bProcessWater:=F_StepCMP(iStep,0,0,0,0,0,0,0,0,0,0);

q_stCmd.bTightAir:=F_StepCMP(iStep,50,100,0,0,0,0,0,0,0,0);
q_stCmd.bChopper1_Air:=F_StepCMP(iStep,0,0,0,0,0,0,0,0,0,0);
q_stCmd.bChopper2_Air:=F_StepCMP(iStep,0,0,0,0,0,0,0,0,0,0);

q_stCmd.bChopper1_Water:=F_StepCMP(iStep,100,0,0,0,0,0,0,0,0,0);
q_stCmd.bChopper2_Water:=F_StepCMP(iStep,100,0,0,0,0,0,0,0,0,0);


//Statistic and Status
tonStepTime(IN:=q_bRunning,PT:=T#5H);
q_tStepTime:=tonStepTime.ET;

END_PROGRAM

// ---- POUs/2. Process/Cleaning/_Control.TcPOU
PROGRAM _Control
VAR_INPUT
	i_bStart						:BOOL;
	i_bStepFinished					:BOOL;
	i_bProcessFinished				:BOOL;
	i_bSkipStep						:BOOL;
END_VAR
VAR
	iStep							:INT;
	tonStepTime						:TON;
END_VAR
VAR_OUTPUT
	q_bRunning						:BOOL;
	q_bFinished						:BOOL;
	q_stCmd							:ST_ProcessCmd;
	q_bReqFlapOpen					:BOOL;
	q_bReqFlapClosed				:BOOL;
	q_tStepTime						:TIME;
END_VAR

q_bRunning:=iStep<>0;

IF i_bSkipStep THEN
	iStep:=1000;
END_IF

IF NOT i_bStart THEN
	iStep:=0;
END_IF

CASE iStep OF
	0:
		IF i_bStart THEN
			q_bFinished:=FALSE;
			iStep:=50;
		END_IF
	
	//Mixer and Choppers are rotating
	50:
		IF i_bProcessFinished THEN
			iStep:=1000;
		END_IF
	
		
	1000:
		q_bFinished:=TRUE;
		IF i_bStepFinished THEN
			iStep:=0;
		END_IF
END_CASE


//Statistic and Status
tonStepTime(IN:=q_bRunning,PT:=T#5H);
q_tStepTime:=tonStepTime.ET;

END_PROGRAM

// ---- POUs/2. Process/P2_03_Production_Ctrl.TcPOU
PROGRAM P2_03_Production_Ctrl
VAR
	bFeeding_Active						:BOOL;
	bMixing_Active						:BOOL;
	bDischarging_Active					:BOOL;
	
	bDischargeCloseRequest				:BOOL;
	bDischargeOpenRequest				:BOOL;
END_VAR
VAR // added by the converter: edge detectors and wires of the graphical bodies
    _w1, _w2, _w3 : BOOL;
END_VAR

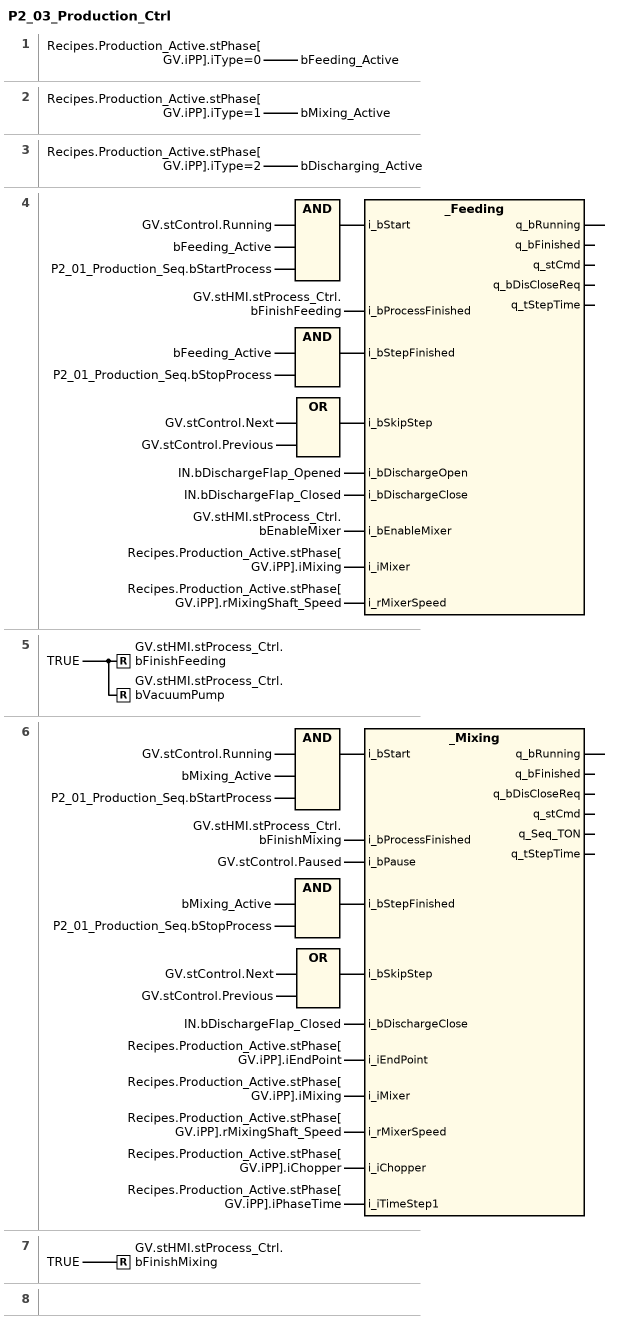
// NETWORK 1
bFeeding_Active := Recipes.Production_Active.stPhase[GV.iPP].iType=0;

// NETWORK 2
bMixing_Active := Recipes.Production_Active.stPhase[GV.iPP].iType=1;

// NETWORK 3
bDischarging_Active := Recipes.Production_Active.stPhase[GV.iPP].iType=2;

// NETWORK 4
_Feeding(i_bStart := GV.stControl.Running AND bFeeding_Active AND P2_01_Production_Seq.bStartProcess, i_bProcessFinished := GV.stHMI.stProcess_Ctrl.bFinishFeeding, i_bStepFinished := bFeeding_Active AND P2_01_Production_Seq.bStopProcess, i_bSkipStep := GV.stControl.Next OR GV.stControl.Previous, i_bDischargeOpen := IN.bDischargeFlap_Opened, i_bDischargeClose := IN.bDischargeFlap_Closed, i_bEnableMixer := GV.stHMI.stProcess_Ctrl.bEnableMixer, i_iMixer := Recipes.Production_Active.stPhase[GV.iPP].iMixing, i_rMixerSpeed := Recipes.Production_Active.stPhase[GV.iPP].rMixingShaft_Speed);

// NETWORK 5
GV.stHMI.stProcess_Ctrl.bFinishFeeding R= TRUE;
GV.stHMI.stProcess_Ctrl.bVacuumPump R= TRUE;

// NETWORK 6
_Mixing(i_bStart := GV.stControl.Running AND bMixing_Active AND P2_01_Production_Seq.bStartProcess, i_bProcessFinished := GV.stHMI.stProcess_Ctrl.bFinishMixing, i_bPause := GV.stControl.Paused, i_bStepFinished := bMixing_Active AND P2_01_Production_Seq.bStopProcess, i_bSkipStep := GV.stControl.Next OR GV.stControl.Previous, i_bDischargeClose := IN.bDischargeFlap_Closed, i_iEndPoint := Recipes.Production_Active.stPhase[GV.iPP].iEndPoint, i_iMixer := Recipes.Production_Active.stPhase[GV.iPP].iMixing, i_rMixerSpeed := Recipes.Production_Active.stPhase[GV.iPP].rMixingShaft_Speed, i_iChopper := Recipes.Production_Active.stPhase[GV.iPP].iChopper, i_iTimeStep1 := Recipes.Production_Active.stPhase[GV.iPP].iPhaseTime);

// NETWORK 7
GV.stHMI.stProcess_Ctrl.bFinishMixing R= TRUE;

// NETWORK 8

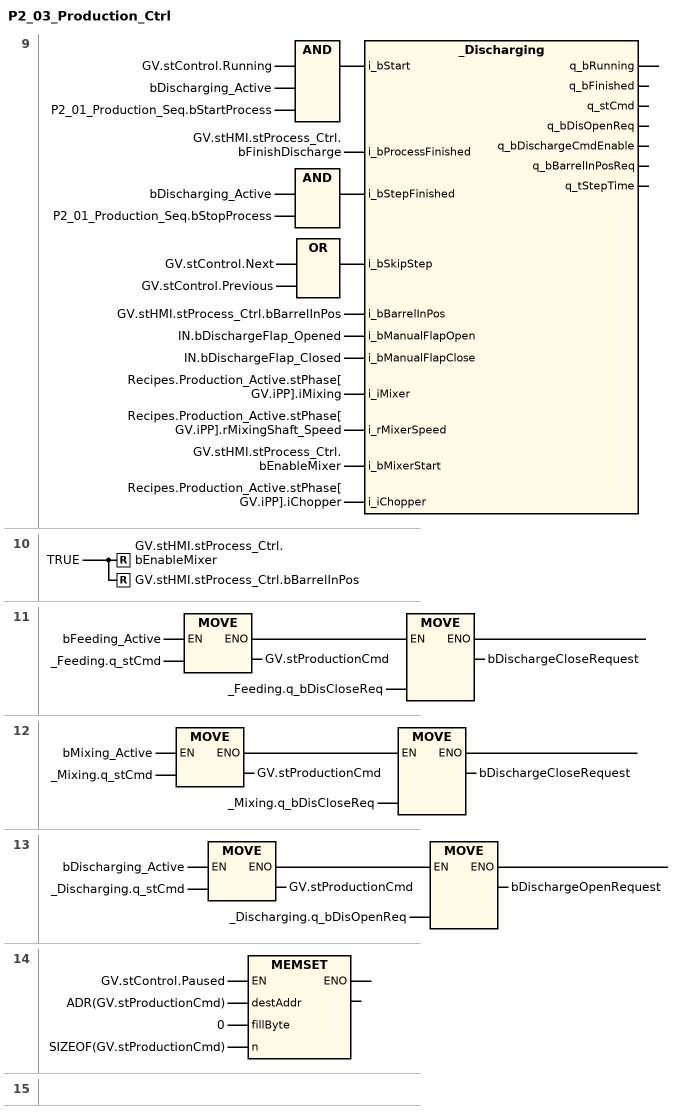
// NETWORK 9
_Discharging(i_bStart := GV.stControl.Running AND bDischarging_Active AND P2_01_Production_Seq.bStartProcess, i_bProcessFinished := GV.stHMI.stProcess_Ctrl.bFinishDischarge, i_bStepFinished := bDischarging_Active AND P2_01_Production_Seq.bStopProcess, i_bSkipStep := GV.stControl.Next OR GV.stControl.Previous, i_bBarrelInPos := GV.stHMI.stProcess_Ctrl.bBarrelInPos, i_bManualFlapOpen := IN.bDischargeFlap_Opened, i_bManualFlapClose := IN.bDischargeFlap_Closed, i_iMixer := Recipes.Production_Active.stPhase[GV.iPP].iMixing, i_rMixerSpeed := Recipes.Production_Active.stPhase[GV.iPP].rMixingShaft_Speed, i_bMixerStart := GV.stHMI.stProcess_Ctrl.bEnableMixer, i_iChopper := Recipes.Production_Active.stPhase[GV.iPP].iChopper);

// NETWORK 10
GV.stHMI.stProcess_Ctrl.bEnableMixer R= TRUE;
GV.stHMI.stProcess_Ctrl.bBarrelInPos R= TRUE;

// NETWORK 11
_w1 := bFeeding_Active;
IF _w1 THEN GV.stProductionCmd := _Feeding.q_stCmd; END_IF
IF _w1 THEN bDischargeCloseRequest := _Feeding.q_bDisCloseReq; END_IF

// NETWORK 12
_w2 := bMixing_Active;
IF _w2 THEN GV.stProductionCmd := _Mixing.q_stCmd; END_IF
IF _w2 THEN bDischargeCloseRequest := _Mixing.q_bDisCloseReq; END_IF

// NETWORK 13
_w3 := bDischarging_Active;
IF _w3 THEN GV.stProductionCmd := _Discharging.q_stCmd; END_IF
IF _w3 THEN bDischargeOpenRequest := _Discharging.q_bDisOpenReq; END_IF

// NETWORK 14
IF GV.stControl.Paused THEN
    MEMSET(destAddr := ADR(GV.stProductionCmd), fillByte := 0, n := SIZEOF(GV.stProductionCmd));
END_IF

// NETWORK 15

END_PROGRAM

// ---- POUs/2. Process/P2_04_Cleaning_Ctrl.TcPOU
PROGRAM P2_04_Cleaning_Ctrl
VAR
	bPreWash_Active					:BOOL;
	bMounting_Active				:BOOL;
	bMainClean_Active				:BOOL;
	bPWClean_Active					:BOOL;
	bRinsing_Active					:BOOL;
	bBlowing_Active					:BOOL;
	bControl_Active					:BOOL;
	
	bDischargeCloseRequest				:BOOL;
	bDischargeOpenRequest				:BOOL;
END_VAR
VAR // added by the converter: edge detectors and wires of the graphical bodies
    _w1, _w2, _w3, _w4 : BOOL;
END_VAR

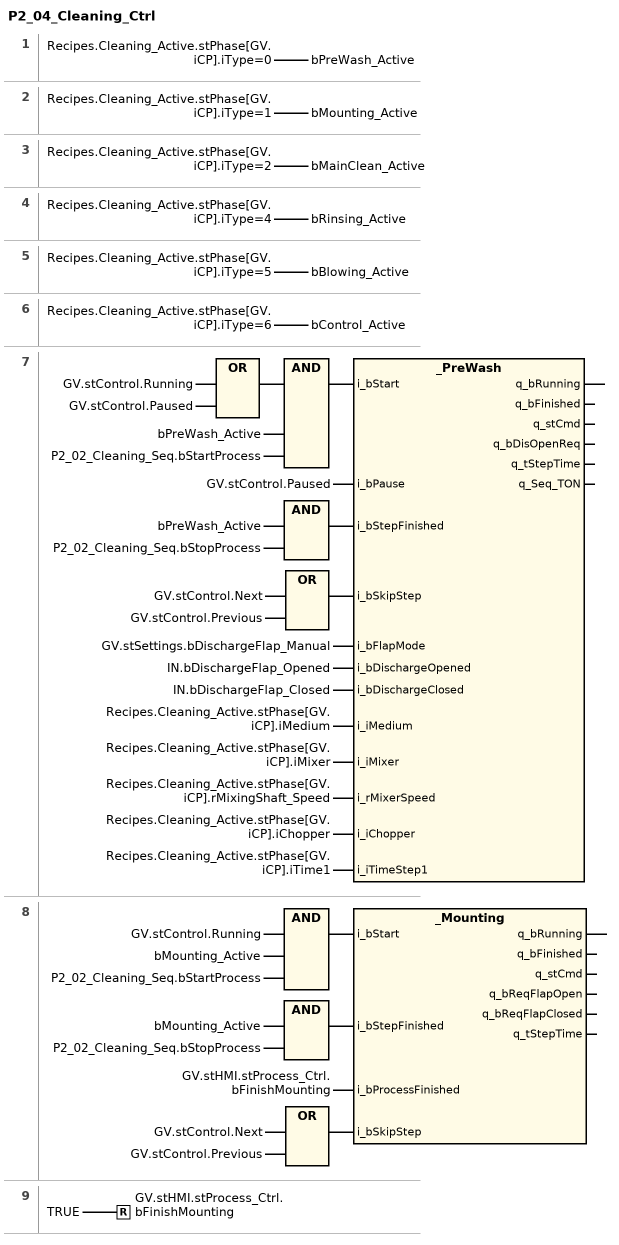
// NETWORK 1
bPreWash_Active := Recipes.Cleaning_Active.stPhase[GV.iCP].iType=0;

// NETWORK 2
bMounting_Active := Recipes.Cleaning_Active.stPhase[GV.iCP].iType=1;

// NETWORK 3
bMainClean_Active := Recipes.Cleaning_Active.stPhase[GV.iCP].iType=2;

// NETWORK 4
bRinsing_Active := Recipes.Cleaning_Active.stPhase[GV.iCP].iType=4;

// NETWORK 5
bBlowing_Active := Recipes.Cleaning_Active.stPhase[GV.iCP].iType=5;

// NETWORK 6
bControl_Active := Recipes.Cleaning_Active.stPhase[GV.iCP].iType=6;

// NETWORK 7
_PreWash(i_bStart := (GV.stControl.Running OR GV.stControl.Paused) AND bPreWash_Active AND P2_02_Cleaning_Seq.bStartProcess, i_bPause := GV.stControl.Paused, i_bStepFinished := bPreWash_Active AND P2_02_Cleaning_Seq.bStopProcess, i_bSkipStep := GV.stControl.Next OR GV.stControl.Previous, i_bFlapMode := GV.stSettings.bDischargeFlap_Manual, i_bDischargeOpened := IN.bDischargeFlap_Opened, i_bDischargeClosed := IN.bDischargeFlap_Closed, i_iMedium := Recipes.Cleaning_Active.stPhase[GV.iCP].iMedium, i_iMixer := Recipes.Cleaning_Active.stPhase[GV.iCP].iMixer, i_rMixerSpeed := Recipes.Cleaning_Active.stPhase[GV.iCP].rMixingShaft_Speed, i_iChopper := Recipes.Cleaning_Active.stPhase[GV.iCP].iChopper, i_iTimeStep1 := Recipes.Cleaning_Active.stPhase[GV.iCP].iTime1);

// NETWORK 8
_Mounting(i_bStart := GV.stControl.Running AND bMounting_Active AND P2_02_Cleaning_Seq.bStartProcess, i_bStepFinished := bMounting_Active AND P2_02_Cleaning_Seq.bStopProcess, i_bProcessFinished := GV.stHMI.stProcess_Ctrl.bFinishMounting, i_bSkipStep := GV.stControl.Next OR GV.stControl.Previous);

// NETWORK 9
GV.stHMI.stProcess_Ctrl.bFinishMounting R= TRUE;

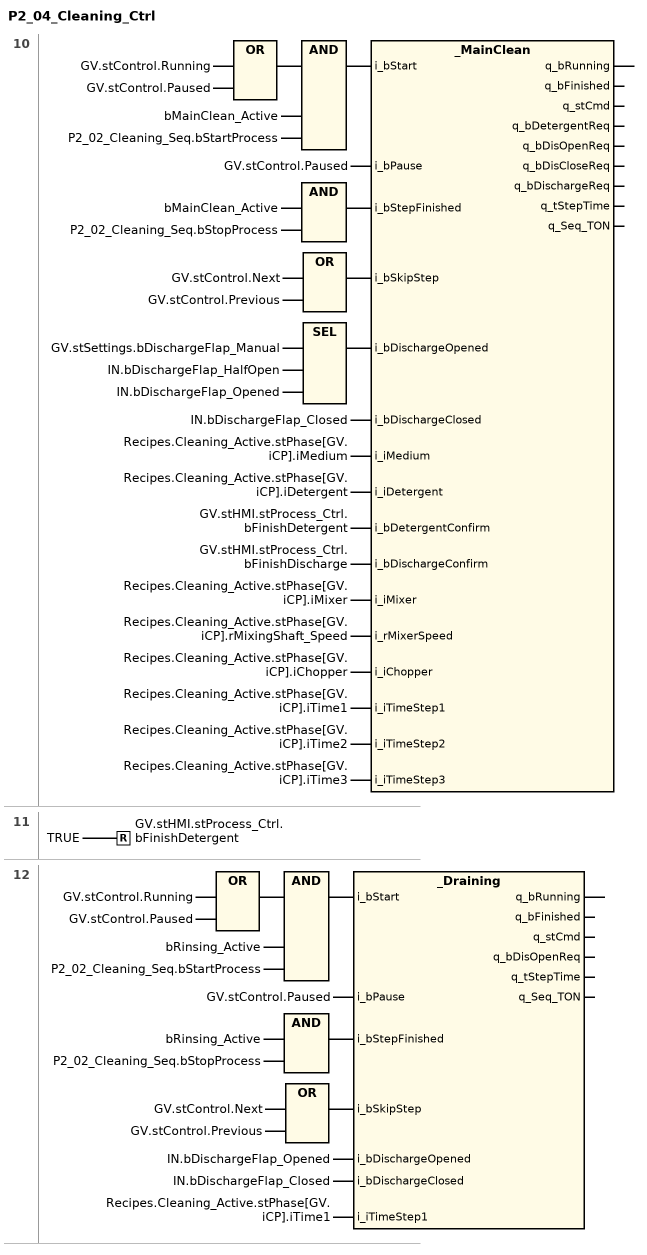
// NETWORK 10
_MainClean(i_bStart := (GV.stControl.Running OR GV.stControl.Paused) AND bMainClean_Active AND P2_02_Cleaning_Seq.bStartProcess, i_bPause := GV.stControl.Paused, i_bStepFinished := bMainClean_Active AND P2_02_Cleaning_Seq.bStopProcess, i_bSkipStep := GV.stControl.Next OR GV.stControl.Previous, i_bDischargeOpened := SEL(GV.stSettings.bDischargeFlap_Manual, IN.bDischargeFlap_HalfOpen, IN.bDischargeFlap_Opened), i_bDischargeClosed := IN.bDischargeFlap_Closed, i_iMedium := Recipes.Cleaning_Active.stPhase[GV.iCP].iMedium, i_iDetergent := Recipes.Cleaning_Active.stPhase[GV.iCP].iDetergent, i_bDetergentConfirm := GV.stHMI.stProcess_Ctrl.bFinishDetergent, i_bDischargeConfirm := GV.stHMI.stProcess_Ctrl.bFinishDischarge, i_iMixer := Recipes.Cleaning_Active.stPhase[GV.iCP].iMixer, i_rMixerSpeed := Recipes.Cleaning_Active.stPhase[GV.iCP].rMixingShaft_Speed, i_iChopper := Recipes.Cleaning_Active.stPhase[GV.iCP].iChopper, i_iTimeStep1 := Recipes.Cleaning_Active.stPhase[GV.iCP].iTime1, i_iTimeStep2 := Recipes.Cleaning_Active.stPhase[GV.iCP].iTime2, i_iTimeStep3 := Recipes.Cleaning_Active.stPhase[GV.iCP].iTime3);

// NETWORK 11
GV.stHMI.stProcess_Ctrl.bFinishDetergent R= TRUE;

// NETWORK 12
_Draining(i_bStart := (GV.stControl.Running OR GV.stControl.Paused) AND bRinsing_Active AND P2_02_Cleaning_Seq.bStartProcess, i_bPause := GV.stControl.Paused, i_bStepFinished := bRinsing_Active AND P2_02_Cleaning_Seq.bStopProcess, i_bSkipStep := GV.stControl.Next OR GV.stControl.Previous, i_bDischargeOpened := IN.bDischargeFlap_Opened, i_bDischargeClosed := IN.bDischargeFlap_Closed, i_iTimeStep1 := Recipes.Cleaning_Active.stPhase[GV.iCP].iTime1);

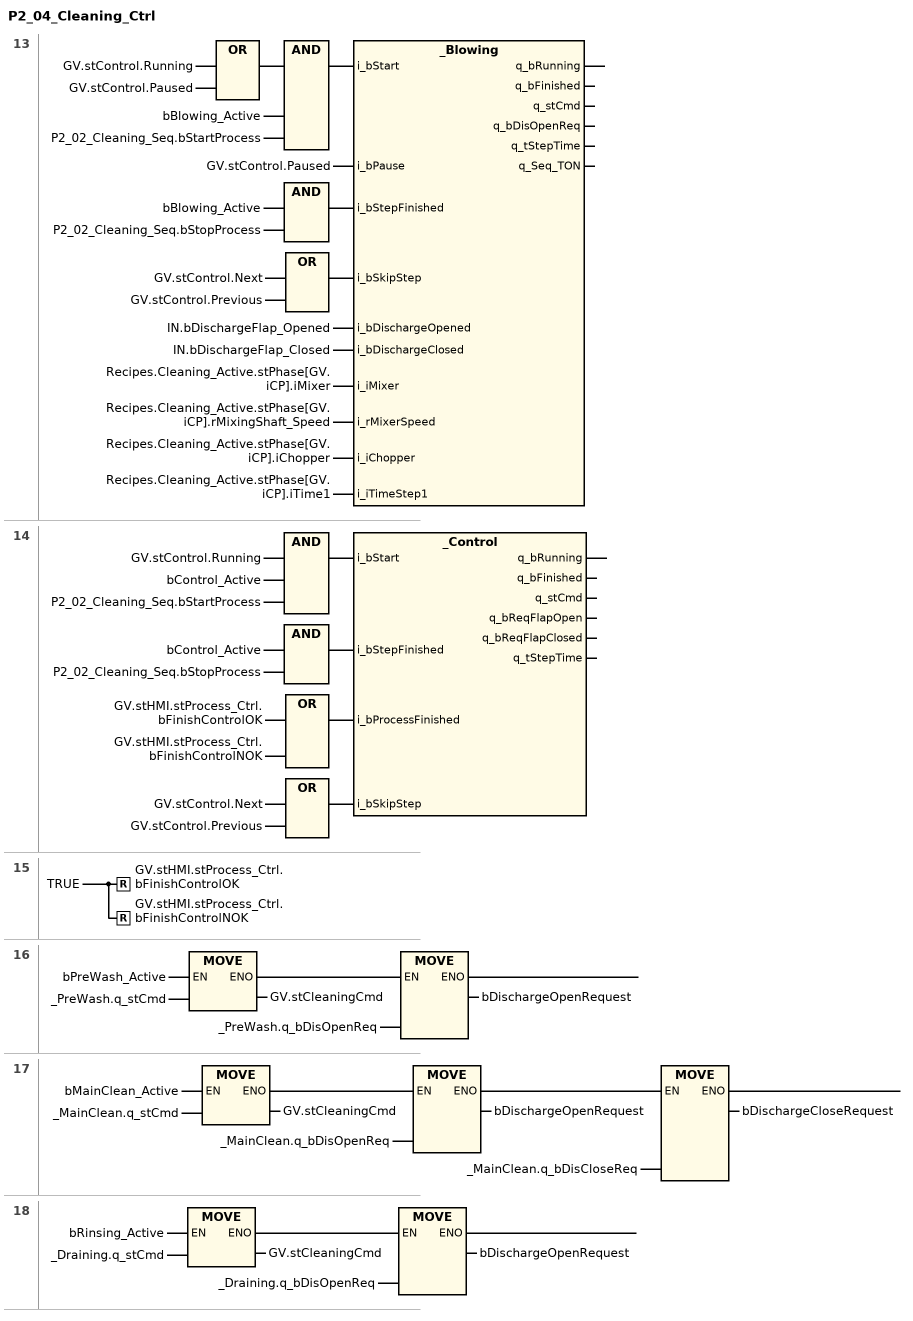
// NETWORK 13
_Blowing(i_bStart := (GV.stControl.Running OR GV.stControl.Paused) AND bBlowing_Active AND P2_02_Cleaning_Seq.bStartProcess, i_bPause := GV.stControl.Paused, i_bStepFinished := bBlowing_Active AND P2_02_Cleaning_Seq.bStopProcess, i_bSkipStep := GV.stControl.Next OR GV.stControl.Previous, i_bDischargeOpened := IN.bDischargeFlap_Opened, i_bDischargeClosed := IN.bDischargeFlap_Closed, i_iMixer := Recipes.Cleaning_Active.stPhase[GV.iCP].iMixer, i_rMixerSpeed := Recipes.Cleaning_Active.stPhase[GV.iCP].rMixingShaft_Speed, i_iChopper := Recipes.Cleaning_Active.stPhase[GV.iCP].iChopper, i_iTimeStep1 := Recipes.Cleaning_Active.stPhase[GV.iCP].iTime1);

// NETWORK 14
_Control(i_bStart := GV.stControl.Running AND bControl_Active AND P2_02_Cleaning_Seq.bStartProcess, i_bStepFinished := bControl_Active AND P2_02_Cleaning_Seq.bStopProcess, i_bProcessFinished := GV.stHMI.stProcess_Ctrl.bFinishControlOK OR GV.stHMI.stProcess_Ctrl.bFinishControlNOK, i_bSkipStep := GV.stControl.Next OR GV.stControl.Previous);

// NETWORK 15
GV.stHMI.stProcess_Ctrl.bFinishControlOK R= TRUE;
GV.stHMI.stProcess_Ctrl.bFinishControlNOK R= TRUE;

// NETWORK 16
_w1 := bPreWash_Active;
IF _w1 THEN GV.stCleaningCmd := _PreWash.q_stCmd; END_IF
IF _w1 THEN bDischargeOpenRequest := _PreWash.q_bDisOpenReq; END_IF

// NETWORK 17
_w2 := bMainClean_Active;
IF _w2 THEN GV.stCleaningCmd := _MainClean.q_stCmd; END_IF
IF _w2 THEN bDischargeOpenRequest := _MainClean.q_bDisOpenReq; END_IF
IF _w2 THEN bDischargeCloseRequest := _MainClean.q_bDisCloseReq; END_IF

// NETWORK 18
_w3 := bRinsing_Active;
IF _w3 THEN GV.stCleaningCmd := _Draining.q_stCmd; END_IF
IF _w3 THEN bDischargeOpenRequest := _Draining.q_bDisOpenReq; END_IF

